// Mitsubishi GX Works2 project: Slave_V37_FERDIG   PLC: FX3U/FX3UC

// global labels: Global1
VAR_GLOBAL
  send_aapning_reg_ventil AT D8262 : INT;  (* ÅPNING REGVENTIL *)
  utstroom_analogt AT D8261 : INT;  (* FLOWMETER *)
  tanknivaa_analogt AT D8260 : INT;  (* NIVÅMÅLER *)
  start_bit AT M101 : BOOL;  (* M100 til M199 Reserveres TIL SLAVE *)
  tvangstyr_startsignal_frekv AT M1 : BOOL;  (* Aktiver kontaktor for startsignal til omformer / M0 til M99 Reservert INTERNT i slave *)
  intern_start_regventil AT M2 : BOOL;
  intern_aktiver_magventil_1 AT M4 : BOOL;  (* Lokalt for slave *)
  intern_aktiver_magventil_2 AT M5 : BOOL;  (* Lokalt for slave *)
  intern_aktiver_magventil_3 AT M6 : BOOL;  (* Lokalt for slave *)
  lest_tanknivaa AT D1 : INT;  (* LAGRING AV WORDS *)
  status_brytere AT D2 : INT;  (* Start,stopp,ACK og AutoModus *)
  referanse AT D5 : INT;
  Td AT D6 : INT;
  Ti AT D7 : INT;
  Kp AT D8 : INT;
  reg_modus AT D9 : INT;  (* 4bit *)
  u0_nompaadrag_fra_scada AT D10 : INT;
  lest_utstroom AT D21 : INT;
END_VAR
VAR_GLOBAL CONSTANT
  start_omformer : INT := 1151;  (* KONSTANTER *)
  stopp_omformer : INT := 1087;
  quickstop_omformer : INT := 1135;
  fult_aapen_regventil : INT := 4000;
  fult_lukket_regventil : INT := 500;
  fult_paadrag_pumpe : INT := 16310;  (* 16310 før skalering *)
END_VAR
VAR_GLOBAL
  fysisk_start_frekomformer AT Y000 : BOOL;  (* K4 / UTGANGER *)
  alarm_lampe AT Y001 : BOOL;  (* Alarmlampe *)
  magnetventil_1 AT Y004 : BOOL;  (* K1 *)
  magnetventil_2 AT Y005 : BOOL;  (* K2 *)
  magnetventil_3 AT Y006 : BOOL;  (* K3 *)
  strømbrudd AT M500 : BOOL;
  kritisk_refnivaa_opnaad_slave AT M202 : BOOL;
  kritiaskalarm_aapne_ventiler AT M203 : BOOL;
  kritiskalarm_nedre_stengventiler AT M206 : BOOL;
  fortsatt_kritisk_nedre AT M207 : BOOL;
  fortsatt_kritisk_oovre AT M208 : BOOL;
  fortsatt_alarm AT M209 : BOOL;
  alarm_oovre AT M300 : BOOL;  (* M300 til M399 beholdes FRA SLAVE *)
  kritiskalarm_oovre AT M301 : BOOL;
  ACK_slave AT M302 : BOOL;
  samplingstid AT D12 : INT;
  tau_lead AT D13 : INT;
  tau_lag AT D14 : INT;
  d_filter AT D15 : INT;
  rate_limit AT D16 : INT;
  tt AT D17 : INT;
  ref_skalert_som_tankmaaling AT D22 : INT;
  stasjonært_avvik AT M303 : BOOL;
END_VAR
VAR_GLOBAL CONSTANT
  hysterese_alarmgrense : INT := 20;
END_VAR
VAR_GLOBAL
  strømbrudd_slave AT M304 : BOOL;
  alarm_nedre AT M305 : BOOL;  (* M300 til M399 beholdes FRA SLAVE *)
  kritiskalarm_nedre AT M306 : BOOL;
  paadrag_manuelt AT D34 : INT;
  kritisk_lav_eller_hooy AT M210 : BOOL;
  stopp AT M201 : BOOL;
  start AT M200 : BOOL;  (* INTERNT I SLAVE *)
  oppstart AT M211 : BOOL;
  auto_ACK AT M212 : BOOL;
  stopp_slave AT M307 : BOOL;
  under_refnivaa AT M213 : BOOL;  (* M213 til M215 *)
  auto_ACK_lav_hooy AT M216 : BOOL;
  frekvenspaadrag_til_omformer AT D33 : INT;
END_VAR
VAR_GLOBAL CONSTANT
  blinkrate : INT := 1;
END_VAR
VAR_GLOBAL
  kfk AT D18 : INT;  (* Foroverkoblingsparameter *)
  forrige_paadrag_regulator AT D52 : REAL;
  tanknivaa_til_regulator AT D40 : REAL;
  u0_nompaadrag_til_regulator AT D46 : REAL;
  paadrag_fra_regulator AT D48 : REAL;
  manuelt_paadrag_til_regulator AT D50 : REAL;
  control_word AT D32 : INT;
  paadrag_til_scada AT D4 : INT;  (* Start,stopp,ACK og AutoModus *)
  tanknivaa_til_scada AT D0 : INT;
  aapning_reg_ventil AT D23 : INT;
  ventil_paadrag AT D36 : INT;
  tanknivaa_filtrert AT D24 : INT;
  stasjonært_avvik_verdi AT D25 : INT;
  paadrag_regulator AT D26 : INT;  (* RegulatorParmarametere *)
  referanse_til_PID AT D42 : REAL;
  magnetventil_1_ACK AT M308 : BOOL;
  magnetventil_2_ACK AT M309 : BOOL;
  magnetventil_3_ACK AT M310 : BOOL;
END_VAR
VAR_GLOBAL CONSTANT
  null_paadrag_pumpe : INT;  (* 16310 før skalering *)
END_VAR
VAR_GLOBAL
  glatt_referanse AT D44 : REAL;
  glatt_referanse_til_scada AT D38 : INT;
  reg_modus_bit AT M112 : BOOL;  (* Til og med M115 *)
  kritisk_lav_eller_hooy_bit AT M111 : BOOL;
  testmodus_bit AT M110 : BOOL;
  anti_windup_bit AT M109 : BOOL;
  forover_kobling_bit AT M108 : BOOL;
  pumpe_regulering_bit AT M107 : BOOL;
  ventil_regulering_bit AT M106 : BOOL;
  aktiver_magv_3_bit AT M105 : BOOL;
  aktiver_magv_2_bit AT M104 : BOOL;
  aktiver_magv_1_bit AT M103 : BOOL;
  ACK_bit AT M102 : BOOL;
  stopp_bit AT M100 : BOOL;
  magnetventil_aapen_igjen AT M311 : BOOL;
  pumpe_regulering AT M312 : BOOL;
  ventil_regulering AT M313 : BOOL;
  Profibus_ok AT M314 : BOOL;
  kritiskalarm_refnivaa_oppnaad AT M315 : BOOL;
  ventil_skalert AT D37 : INT;
  utstroom_filtrert AT D20 : INT;
  frk_control AT M400 : BOOL;  (* Høy = klar, Lav = ikke klar / Statusmeldinger fra frekvensomformeren *)
  frk_VLT AT M401 : BOOL;
  frk_motor_coasting AT M402 : BOOL;
  frk_trip AT M403 : BOOL;
  frk_on_2 AT M404 : BOOL;
  frk_on_3 AT M405 : BOOL;
  frk_stop_enable AT M406 : BOOL;
  frk_warning AT M407 : BOOL;
  frk_speed_ref AT M408 : BOOL;
  frk_local_operation AT M409 : BOOL;
  frk_frequency_ok AT M410 : BOOL;
  frk_running AT M411 : BOOL;
  frk_spenning_ok AT M413 : BOOL;
  frk_moment_ok AT M414 : BOOL;
  frk_termisk_varsel AT M415 : BOOL;
  testmode_ACK AT M316 : BOOL;
  utstroom_til_regulator AT D54 : REAL;
  utstroom_til_scada AT D39 : INT;
  ubrukt_2 AT D100 : INT;
  ubrukt_3 AT D101 : INT;
  ubrukt_4 AT D102 : INT;
  ubrukt_15 AT D103 : INT;
  innenfor_refomraade AT M214 : BOOL;  (* M213 til M215 *)
  over_refnivaa AT M215 : BOOL;  (* M213 til M215 *)
  reg_modus_ACK AT M317 : BOOL;  (* M317 til og med M320 *)
  under_60_nivaa AT M217 : BOOL;
  frekvens_skalert AT D35 : INT;
END_VAR

// task Task_01 (event TRUE, interval 0, priority 31): POU_01
// task task_2 (event FALSE, interval T#200ms, priority 31): Regulator
// task stroombrudd (event TRUE, interval 0, priority 31): stroombrudd

PROGRAM POU_01
VAR
  lavpass_filter_1 : lavpass_filter_tanknivaa;
  lavpass_filter_2 : lavpass_filter_utstrøm;
  DEROUND_1 : DEROUND;
  DEROUND_2 : DEROUND;
  Lampe_Alarm_1 : Lampe_Alarm;
  DEROUND_3 : DEROUND;
  DEROUND_4 : DEROUND;
  DEROUND_5 : DEROUND;
  DEROUND_6 : DEROUND;
  DEROUND_7 : DEROUND;
  skalering_tanknivaa_1 : skalering_tanknivaa;
  skalering_ventil_1 : skalering_ventil;
  skalering_paadrag_1 : skalering_paadrag;
  skalering_referanse_1 : skalering_referanse;
  utregning_stasjonært_avvik_1 : utregning_stasjonært_avvik;
  skalering_til_bruker_ven_og_omf1 : skalering_til_bruker_ven_og_omf;
  skalering_utstroom_1 : skalering_utstroom;
  mottak_av_data_fra_master_1 : mottak_av_data_fra_master;
  sending_av_data_til_master_1 : sending_av_data_til_master;
  kvittering_av_alarmer_1 : kvittering_av_alarmer;
  utganger_1 : utganger;
  kritisk_refnivaa_oppnaad_1 : kritisk_refnivaa_oppnaad;
  reguleringsmodus_1 : reguleringsmodus;
  handling_ved_kritisk_alarm_1 : handling_ved_kritisk_alarm;
  alarmgrenser_1 : alarmgrenser;
END_VAR
(* structured ladder/FBD written out as ST: instructions are called as NAME(EN, inputs, outputs); _pN, _eN, _tN stand for wires *)
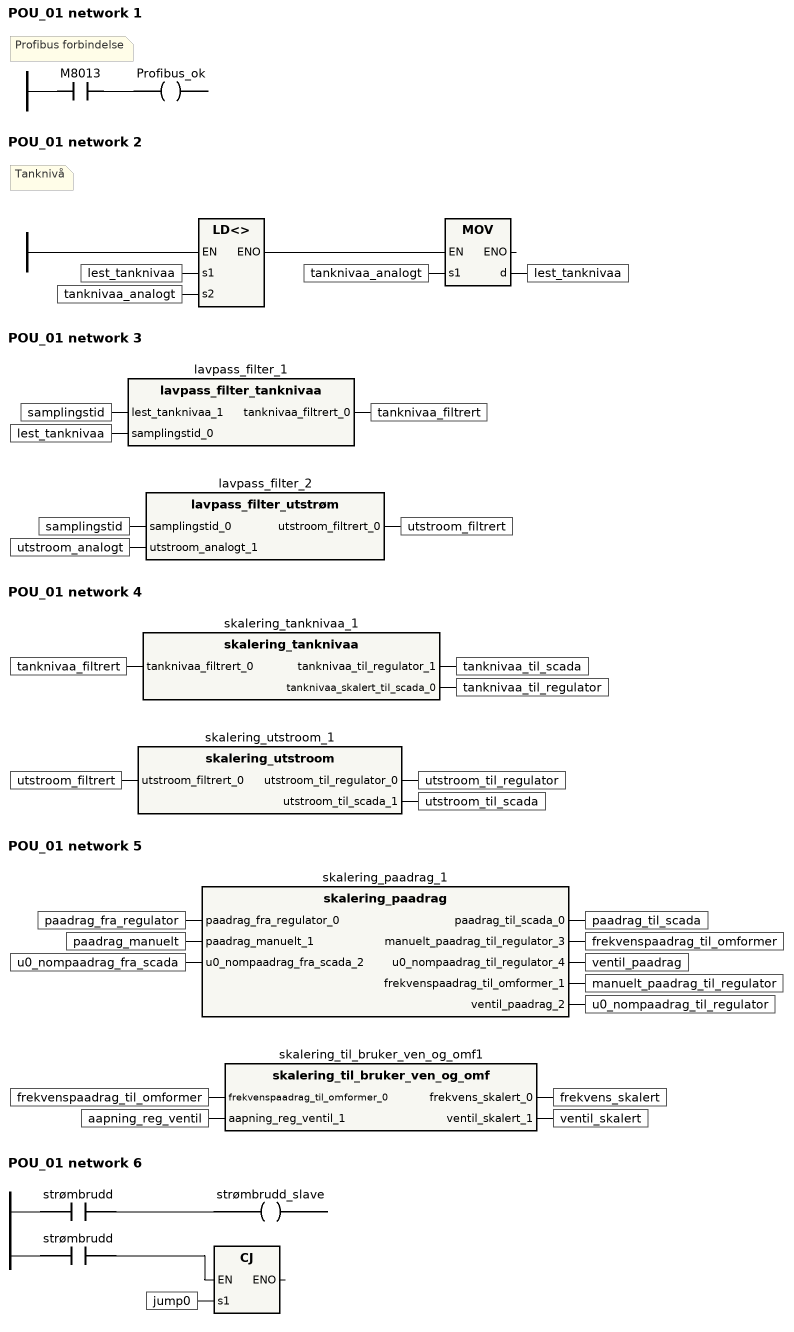
(* network 1 *)
(* Profibus forbindelse *)
Profibus_ok := M8013;
(* network 2 *)
(* Tanknivå *)
_e1 := LD<>(TRUE, lest_tanknivaa, tanknivaa_analogt);
MOV(_e1, tanknivaa_analogt, lest_tanknivaa);
(* network 3 *)
lavpass_filter_1(lest_tanknivaa_1 := samplingstid, samplingstid_0 := lest_tanknivaa, tanknivaa_filtrert_0 => tanknivaa_filtrert);
lavpass_filter_2(samplingstid_0 := samplingstid, utstroom_analogt_1 := utstroom_analogt, utstroom_filtrert_0 => utstroom_filtrert);
(* network 4 *)
skalering_tanknivaa_1(tanknivaa_filtrert_0 := tanknivaa_filtrert, tanknivaa_til_regulator_1 => tanknivaa_til_scada, tanknivaa_skalert_til_scada_0 => tanknivaa_til_regulator);
skalering_utstroom_1(utstroom_filtrert_0 := utstroom_filtrert, utstroom_til_regulator_0 => utstroom_til_regulator, utstroom_til_scada_1 => utstroom_til_scada);
(* network 5 *)
skalering_paadrag_1(paadrag_fra_regulator_0 := paadrag_fra_regulator, paadrag_manuelt_1 := paadrag_manuelt, u0_nompaadrag_fra_scada_2 := u0_nompaadrag_fra_scada, paadrag_til_scada_0 => paadrag_til_scada, manuelt_paadrag_til_regulator_3 => frekvenspaadrag_til_omformer, u0_nompaadrag_til_regulator_4 => ventil_paadrag, frekvenspaadrag_til_omformer_1 => manuelt_paadrag_til_regulator, ventil_paadrag_2 => u0_nompaadrag_til_regulator);
skalering_til_bruker_ven_og_omf1(frekvenspaadrag_til_omformer_0 := frekvenspaadrag_til_omformer, aapning_reg_ventil_1 := aapning_reg_ventil, frekvens_skalert_0 => frekvens_skalert, ventil_skalert_1 => ventil_skalert);
(* network 6 *)
strømbrudd_slave := strømbrudd;
CJ(strømbrudd, jump0);
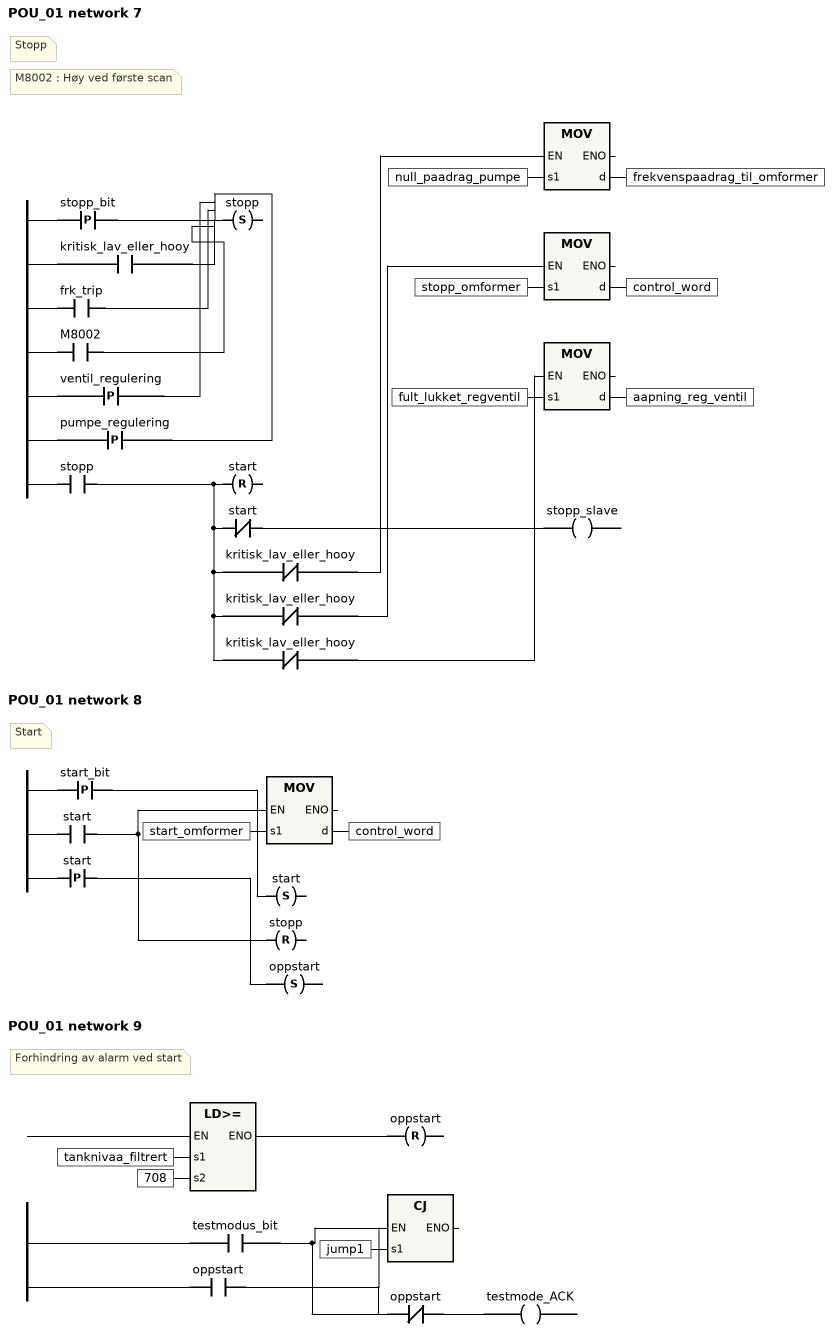
(* network 7 *)
(* Stopp *)
(* M8002 : Høy ved første scan *)
SET(LDP(TRUE, stopp_bit) OR kritisk_lav_eller_hooy OR frk_trip OR M8002 OR LDP(TRUE, ventil_regulering) OR LDP(TRUE, pumpe_regulering), stopp);
RST(stopp, start);
stopp_slave := stopp AND NOT start;
MOV(stopp AND NOT kritisk_lav_eller_hooy, null_paadrag_pumpe, frekvenspaadrag_til_omformer);
MOV(stopp AND NOT kritisk_lav_eller_hooy, stopp_omformer, control_word);
MOV(stopp AND NOT kritisk_lav_eller_hooy, fult_lukket_regventil, aapning_reg_ventil);
(* network 8 *)
(* Start *)
SET(LDP(TRUE, start_bit), start);
RST(start, stopp);
MOV(start, start_omformer, control_word);
SET(LDP(TRUE, start), oppstart);
(* network 9 *)
(* Forhindring av alarm ved start *)
_e1 := LD>=(TRUE, tanknivaa_filtrert, 708);
RST(_e1, oppstart);
_p2 := testmodus_bit OR oppstart;
testmode_ACK := _p2 AND NOT oppstart;
CJ(_p2, jump1);
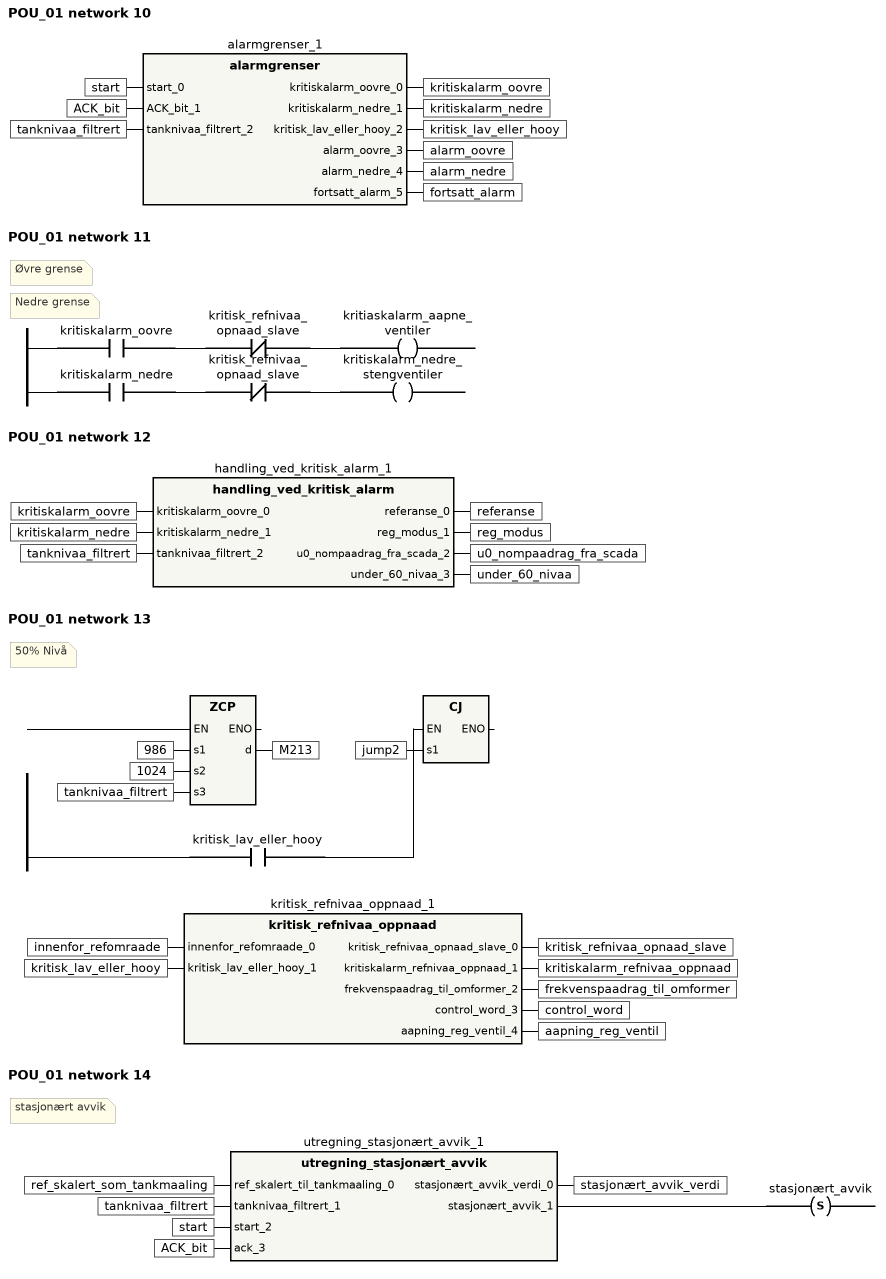
(* network 10 *)
alarmgrenser_1(start_0 := start, ACK_bit_1 := ACK_bit, tanknivaa_filtrert_2 := tanknivaa_filtrert, kritiskalarm_oovre_0 => kritiskalarm_oovre, kritiskalarm_nedre_1 => kritiskalarm_nedre, kritisk_lav_eller_hooy_2 => kritisk_lav_eller_hooy, alarm_oovre_3 => alarm_oovre, alarm_nedre_4 => alarm_nedre, fortsatt_alarm_5 => fortsatt_alarm);
(* network 11 *)
(* Øvre grense *)
(* Nedre grense *)
kritiaskalarm_aapne_ventiler := kritiskalarm_oovre AND NOT kritisk_refnivaa_opnaad_slave;
kritiskalarm_nedre_stengventiler := kritiskalarm_nedre AND NOT kritisk_refnivaa_opnaad_slave;
(* network 12 *)
handling_ved_kritisk_alarm_1(kritiskalarm_oovre_0 := kritiskalarm_oovre, kritiskalarm_nedre_1 := kritiskalarm_nedre, tanknivaa_filtrert_2 := tanknivaa_filtrert, referanse_0 => referanse, reg_modus_1 => reg_modus, u0_nompaadrag_fra_scada_2 => u0_nompaadrag_fra_scada, under_60_nivaa_3 => under_60_nivaa);
(* network 13 *)
(* 50% Nivå *)
ZCP(TRUE, 986, 1024, tanknivaa_filtrert, M213);
kritisk_refnivaa_oppnaad_1(innenfor_refomraade_0 := innenfor_refomraade, kritisk_lav_eller_hooy_1 := kritisk_lav_eller_hooy, kritisk_refnivaa_opnaad_slave_0 => kritisk_refnivaa_opnaad_slave, kritiskalarm_refnivaa_oppnaad_1 => kritiskalarm_refnivaa_oppnaad, frekvenspaadrag_til_omformer_2 => frekvenspaadrag_til_omformer, control_word_3 => control_word, aapning_reg_ventil_4 => aapning_reg_ventil);
CJ(kritisk_lav_eller_hooy, jump2);
(* network 14 *)
(* stasjonært avvik *)
utregning_stasjonært_avvik_1(ref_skalert_til_tankmaaling_0 := ref_skalert_som_tankmaaling, tanknivaa_filtrert_1 := tanknivaa_filtrert, start_2 := start, ack_3 := ACK_bit, stasjonært_avvik_verdi_0 => stasjonært_avvik_verdi);
SET(utregning_stasjonært_avvik_1.stasjonært_avvik_1, stasjonært_avvik);
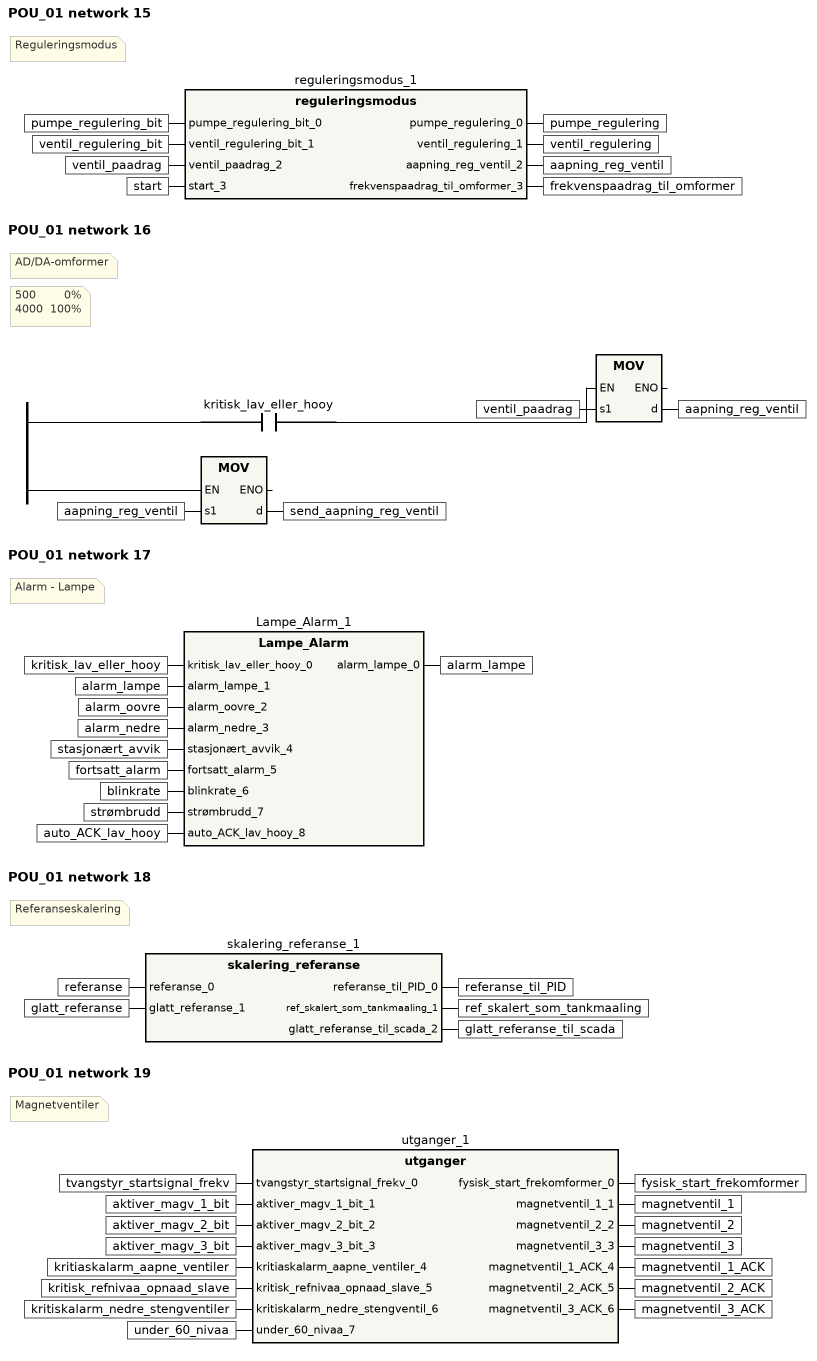
(* network 15 jump1: *)
(* Reguleringsmodus *)
reguleringsmodus_1(pumpe_regulering_bit_0 := pumpe_regulering_bit, ventil_regulering_bit_1 := ventil_regulering_bit, ventil_paadrag_2 := ventil_paadrag, start_3 := start, pumpe_regulering_0 => pumpe_regulering, ventil_regulering_1 => ventil_regulering, aapning_reg_ventil_2 => aapning_reg_ventil, frekvenspaadrag_til_omformer_3 => frekvenspaadrag_til_omformer);
(* network 16 jump2: *)
(* AD/DA-omformer *)
(* 500        0% / 4000  100% *)
MOV(kritisk_lav_eller_hooy, ventil_paadrag, aapning_reg_ventil);
MOV(TRUE, aapning_reg_ventil, send_aapning_reg_ventil);
(* network 17 *)
(* Alarm - Lampe *)
Lampe_Alarm_1(kritisk_lav_eller_hooy_0 := kritisk_lav_eller_hooy, alarm_lampe_1 := alarm_lampe, alarm_oovre_2 := alarm_oovre, alarm_nedre_3 := alarm_nedre, stasjonært_avvik_4 := stasjonært_avvik, fortsatt_alarm_5 := fortsatt_alarm, blinkrate_6 := blinkrate, strømbrudd_7 := strømbrudd, auto_ACK_lav_hooy_8 := auto_ACK_lav_hooy, alarm_lampe_0 => alarm_lampe);
(* network 18 *)
(* Referanseskalering *)
skalering_referanse_1(referanse_0 := referanse, glatt_referanse_1 := glatt_referanse, referanse_til_PID_0 => referanse_til_PID, ref_skalert_som_tankmaaling_1 => ref_skalert_som_tankmaaling, glatt_referanse_til_scada_2 => glatt_referanse_til_scada);
(* network 19 *)
(* Magnetventiler *)
utganger_1(tvangstyr_startsignal_frekv_0 := tvangstyr_startsignal_frekv, aktiver_magv_1_bit_1 := aktiver_magv_1_bit, aktiver_magv_2_bit_2 := aktiver_magv_2_bit, aktiver_magv_3_bit_3 := aktiver_magv_3_bit, kritiaskalarm_aapne_ventiler_4 := kritiaskalarm_aapne_ventiler, kritisk_refnivaa_opnaad_slave_5 := kritisk_refnivaa_opnaad_slave, kritiskalarm_nedre_stengventil_6 := kritiskalarm_nedre_stengventiler, under_60_nivaa_7 := under_60_nivaa, fysisk_start_frekomformer_0 => fysisk_start_frekomformer, magnetventil_1_1 => magnetventil_1, magnetventil_2_2 => magnetventil_2, magnetventil_3_3 => magnetventil_3, magnetventil_1_ACK_4 => magnetventil_1_ACK, magnetventil_2_ACK_5 => magnetventil_2_ACK, magnetventil_3_ACK_6 => magnetventil_3_ACK);
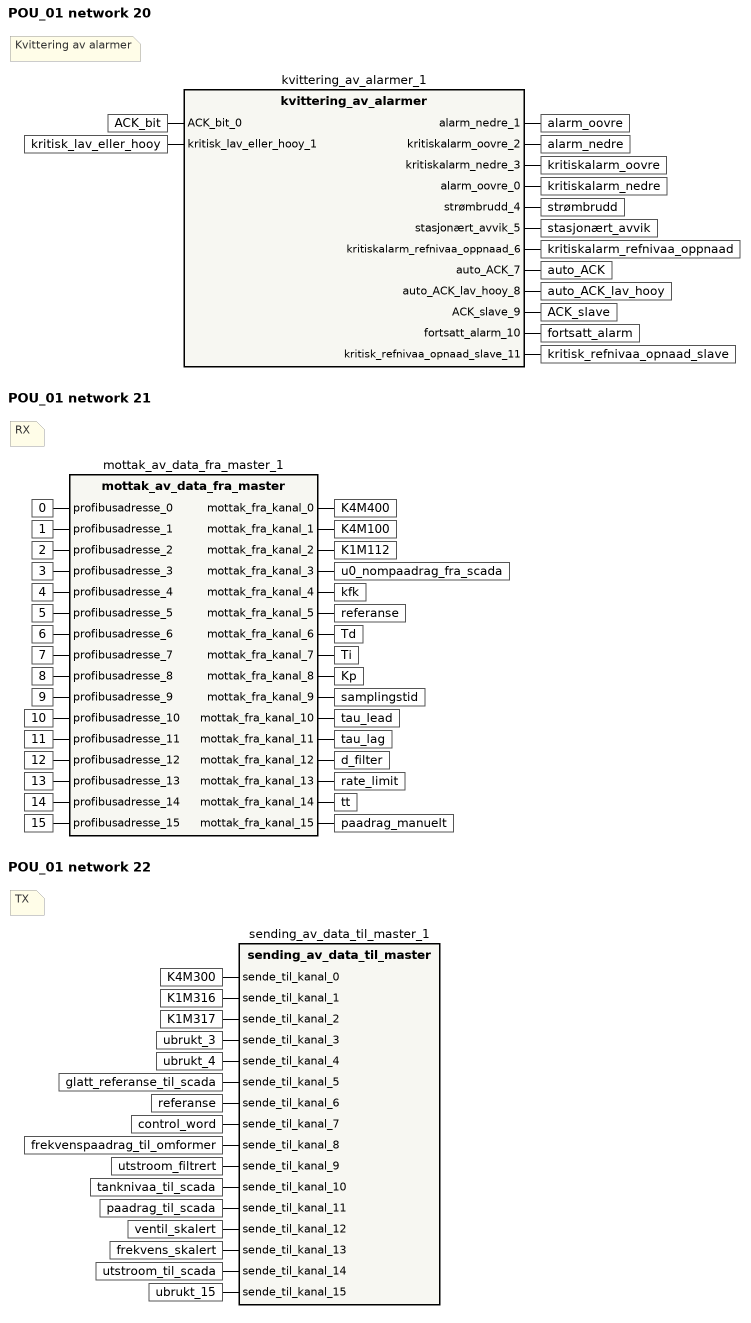
(* network 20 jump0: *)
(* Kvittering av alarmer *)
kvittering_av_alarmer_1(ACK_bit_0 := ACK_bit, kritisk_lav_eller_hooy_1 := kritisk_lav_eller_hooy, alarm_nedre_1 => alarm_oovre, kritiskalarm_oovre_2 => alarm_nedre, kritiskalarm_nedre_3 => kritiskalarm_oovre, alarm_oovre_0 => kritiskalarm_nedre, strømbrudd_4 => strømbrudd, stasjonært_avvik_5 => stasjonært_avvik, kritiskalarm_refnivaa_oppnaad_6 => kritiskalarm_refnivaa_oppnaad, auto_ACK_7 => auto_ACK, auto_ACK_lav_hooy_8 => auto_ACK_lav_hooy, ACK_slave_9 => ACK_slave, fortsatt_alarm_10 => fortsatt_alarm, kritisk_refnivaa_opnaad_slave_11 => kritisk_refnivaa_opnaad_slave);
(* network 21 *)
(* RX *)
mottak_av_data_fra_master_1(profibusadresse_0 := 0, profibusadresse_1 := 1, profibusadresse_2 := 2, profibusadresse_3 := 3, profibusadresse_4 := 4, profibusadresse_5 := 5, profibusadresse_6 := 6, profibusadresse_7 := 7, profibusadresse_8 := 8, profibusadresse_9 := 9, profibusadresse_10 := 10, profibusadresse_11 := 11, profibusadresse_12 := 12, profibusadresse_13 := 13, profibusadresse_14 := 14, profibusadresse_15 := 15, mottak_fra_kanal_0 => K4M400, mottak_fra_kanal_1 => K4M100, mottak_fra_kanal_2 => K1M112, mottak_fra_kanal_3 => u0_nompaadrag_fra_scada, mottak_fra_kanal_4 => kfk, mottak_fra_kanal_5 => referanse, mottak_fra_kanal_6 => Td, mottak_fra_kanal_7 => Ti, mottak_fra_kanal_8 => Kp, mottak_fra_kanal_9 => samplingstid, mottak_fra_kanal_10 => tau_lead, mottak_fra_kanal_11 => tau_lag, mottak_fra_kanal_12 => d_filter, mottak_fra_kanal_13 => rate_limit, mottak_fra_kanal_14 => tt, mottak_fra_kanal_15 => paadrag_manuelt);
(* network 22 *)
(* TX *)
sending_av_data_til_master_1(sende_til_kanal_0 := K4M300, sende_til_kanal_1 := K1M316, sende_til_kanal_2 := K1M317, sende_til_kanal_3 := ubrukt_3, sende_til_kanal_4 := ubrukt_4, sende_til_kanal_5 := glatt_referanse_til_scada, sende_til_kanal_6 := referanse, sende_til_kanal_7 := control_word, sende_til_kanal_8 := frekvenspaadrag_til_omformer, sende_til_kanal_9 := utstroom_filtrert, sende_til_kanal_10 := tanknivaa_til_scada, sende_til_kanal_11 := paadrag_til_scada, sende_til_kanal_12 := ventil_skalert, sende_til_kanal_13 := frekvens_skalert, sende_til_kanal_14 := utstroom_til_scada, sende_til_kanal_15 := ubrukt_15);
END_PROGRAM

FUNCTION_BLOCK lavpass_filter_tanknivaa
VAR CONSTANT
  omega_0 : REAL := 0.2;  (* cutoff frekvens. 16.4: 0.25 mye støy?? gamle:0.0384 *)
  two_pi : REAL := 6.28;  (* 2*pi *)
END_VAR
VAR
  input_float : REAL;
  avg_maaling : REAL;
  avg_maaling_k_minus_1 : REAL;
  filter_faktor : REAL;
  eksponent : REAL;
  tastetid_float : REAL;
END_VAR
VAR_INPUT
  lest_tanknivaa_1 : INT;
END_VAR
VAR_OUTPUT
  tanknivaa_filtrert_0 : INT;
END_VAR
VAR_INPUT
  samplingstid_0 : INT;
END_VAR
VAR
  DEROUND_1 : DEROUND;
END_VAR
tastetid_float :=  INT_TO_REAL (samplingstid_0)/100.0;
eksponent := -tastetid_float*omega_0*two_pi;
filter_faktor := EXP(eksponent);
input_float := INT_TO_REAL (lest_tanknivaa_1);
avg_maaling := filter_faktor * avg_maaling_k_minus_1 + (1.0 - filter_faktor) * input_float;
avg_maaling_k_minus_1 := avg_maaling;
DEROUND_1(real_to_round := avg_maaling, gjelende_siffer_input := 0);
tanknivaa_filtrert_0 := REAL_TO_INT(DEROUND_1.real_rounded);
END_FUNCTION_BLOCK

FUNCTION_BLOCK DEROUND
VAR_INPUT
  real_to_round : REAL;
  gjelende_siffer_input : INT;
END_VAR
VAR
  gjelende_siffer_real : REAL;
  ti_til_gjellende_siffer : REAL;
  int_round : DINT;
END_VAR
VAR_OUTPUT
  real_rounded : REAL;
END_VAR
gjelende_siffer_real := INT_TO_REAL(gjelende_siffer_input);
ti_til_gjellende_siffer := EXP(gjelende_siffer_real * LN(10.0));

IF DINT_TO_REAL(REAL_TO_DINT(real_to_round* ti_til_gjellende_siffer) ) > (real_to_round*ti_til_gjellende_siffer - 0.5) THEN;
	int_round := REAL_TO_DINT(real_to_round * ti_til_gjellende_siffer);
	real_rounded := DINT_TO_REAL(int_round)/ti_til_gjellende_siffer;
ELSE
	int_round := REAL_TO_DINT(real_to_round * ti_til_gjellende_siffer + 1.0);
	real_rounded := DINT_TO_REAL(int_round)/ti_til_gjellende_siffer;
END_IF;
END_FUNCTION_BLOCK

FUNCTION_BLOCK Lampe_Alarm
VAR_OUTPUT
  alarm_lampe_0 : BOOL;
END_VAR
VAR_INPUT
  kritisk_lav_eller_hooy_0 : BOOL;
  alarm_lampe_1 : BOOL;
  alarm_oovre_2 : BOOL;
  alarm_nedre_3 : BOOL;
  stasjonært_avvik_4 : BOOL;
  fortsatt_alarm_5 : BOOL;
  blinkrate_6 : INT;
  strømbrudd_7 : BOOL;
  auto_ACK_lav_hooy_8 : BOOL;
END_VAR
VAR
  lampe_5HZ : BOOL;
  lampe_1HZ : BOOL;
  lampe_konstant : BOOL;
END_VAR
(* structured ladder/FBD written out as ST: instructions are called as NAME(EN, inputs, outputs); _pN, _eN, _tN stand for wires *)
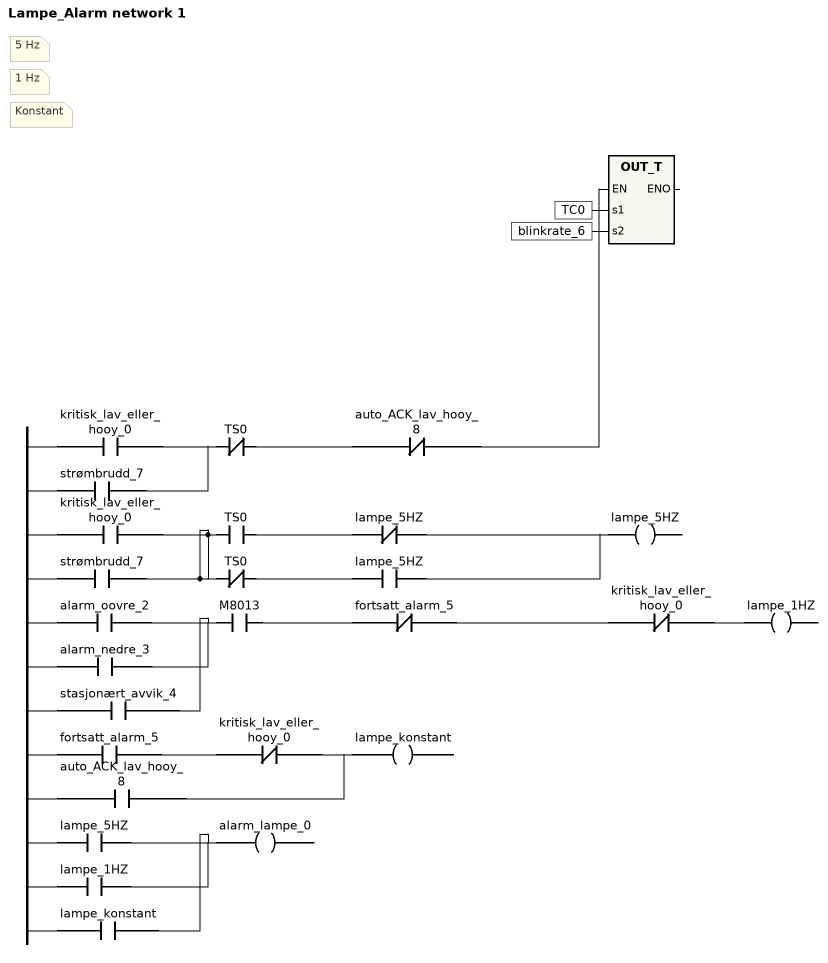
(* network 1 *)
(* 5 Hz *)
(* 1 Hz *)
(* Konstant *)
OUT_T(((kritisk_lav_eller_hooy_0 OR strømbrudd_7) AND NOT TS0) AND NOT auto_ACK_lav_hooy_8, TC0, blinkrate_6);
_p1 := kritisk_lav_eller_hooy_0 OR strømbrudd_7;
lampe_5HZ := (_p1 AND TS0 AND NOT lampe_5HZ) OR (_p1 AND NOT TS0 AND lampe_5HZ);
lampe_1HZ := (((alarm_oovre_2 OR alarm_nedre_3 OR stasjonært_avvik_4) AND M8013) AND NOT fortsatt_alarm_5) AND NOT kritisk_lav_eller_hooy_0;
lampe_konstant := (fortsatt_alarm_5 AND NOT kritisk_lav_eller_hooy_0) OR auto_ACK_lav_hooy_8;
alarm_lampe_0 := lampe_5HZ OR lampe_1HZ OR lampe_konstant;
END_FUNCTION_BLOCK

FUNCTION_BLOCK Lead_lag
VAR_OUTPUT
  u_fk : REAL;
END_VAR
VAR_INPUT
  Kf : INT;  (* random konstant per nå *)
END_VAR
VAR
  forstyrr : REAL;  (* forstyrrelse *)
END_VAR
VAR_INPUT
  Tlead : INT;  (* random konstant per nå *)
  Tlag : INT;  (* random konstant per nå *)
END_VAR
VAR
  last_v : REAL;
END_VAR
VAR_INPUT
  Ts : INT;
END_VAR
VAR
  last_u_fk : REAL;
END_VAR
VAR_INPUT
  leadlag : BOOL;
END_VAR
VAR
  Kf_ny : REAL;
  Tlead_ny : REAL;
  Tlag_ny : REAL;
  Ts_ut : REAL;
END_VAR
VAR_INPUT
  reset : BOOL;
  y_1 : REAL;
  outflow : REAL;
END_VAR
VAR
  forstyrr_ny : REAL;
END_VAR
IF (reset) THEN
	last_v := 0.0;
	last_u_fk := 0.0;
END_IF;

(*Trengs det skalering??*)
Kf_ny := INT_TO_REAL(Kf)/100.00;
Tlead_ny := INT_TO_REAL(Tlead)/100.00;
Tlag_ny := INT_TO_REAL(Tlag)/100.00;
Ts_ut := INT_TO_REAL(Ts)/100.00;

forstyrr := outflow - 0.00025367*y_1*y_1*y_1+0.04313578*y_1*y_1-2.8730536*y_1-5.08111888;

IF forstyrr < 0.00 THEN
	forstyrr_ny := 0.00;
ELSE
	forstyrr_ny := forstyrr;
END_IF;


IF (leadlag=1) THEN
	u_fk := (Kf_ny*Tlead_ny*(forstyrr_ny-last_v)+Kf_ny*forstyrr_ny*Ts_ut+Tlag_ny*last_u_fk)/(Ts_ut+Tlag_ny); 
	(*ingen tidsforsinkelse her, skal vi ha det??*)
	last_v := forstyrr_ny;
	last_u_fk := u_fk;
ELSE
	u_fk := 0.00;
	last_u_fk := 0.00;
END_IF;
END_FUNCTION_BLOCK

FUNCTION_BLOCK PID_regulator
VAR
  last_y : REAL;
END_VAR
VAR_INPUT
  Ts : INT;  (* 0.04 *)
END_VAR
VAR
  up : REAL;
  ud : REAL;
END_VAR
VAR_OUTPUT
  ui : REAL;
END_VAR
VAR
  e_reg : REAL;
  alpha : REAL;
  beta : REAL;
  last_ui : REAL;
  last_ud : REAL;
  last_up : REAL;
END_VAR
VAR_INPUT
  ni : INT;  (* mulig dette skal være input fra intouch idk. *)
  Kp_reg : INT;
  Ti_reg : INT;
  Td_reg : INT;
  r_1 : REAL;
END_VAR
VAR_OUTPUT
  u_ut : REAL;  (* endre til word *)
END_VAR
VAR_INPUT
  y_1 : REAL;
  manual_input : REAL;  (* endre til word *)
  Regulator_type : INT;
  u_fk : REAL;
  u_antiwindup : REAL;
END_VAR
VAR
  Kp_ut : REAL;
  Ti_ut : REAL;
  Td_ut : REAL;
END_VAR
VAR_OUTPUT
  last_u : REAL;
END_VAR
VAR_INPUT
  ratebegrensing : INT;  (* initial value = 2 *)
END_VAR
VAR
  Ts_ut : REAL;
  d_filt : REAL;
  u_reg : REAL;
END_VAR
VAR_INPUT
  reset : BOOL;
  u_it : REAL;
END_VAR
VAR_OUTPUT
  u_t : REAL;
END_VAR
VAR_INPUT
  u_rykkfri : REAL;
END_VAR
VAR
  last_u_nom : REAL;
END_VAR
VAR_INPUT
  u_nominel : REAL;
END_VAR
VAR
  u_nom : REAL;
  konstant : REAL;
END_VAR
IF (reset) THEN
	last_up := 0.0;
	last_ui := 0.0;
	last_ud := 0.0;
	last_y := 0.0;
	last_u_nom := 0.00;
END_IF;

Kp_ut := INT_TO_REAL(Kp)/100.00;
Ti_ut := INT_TO_REAL(Ti)/100.00; 
Td_ut := INT_TO_REAL(Td)/100.00;
Ts_ut := INT_TO_REAL(Ts)/100.00;
d_filt := INT_TO_REAL(ni)/100.00; 

e_reg := r_1-y_1;

alpha := Ts_ut / Ti_ut;
beta :=  Td_ut/(Td_ut+d_filt*Ts_ut);

up := e_reg*Kp_ut;

IF (up-last_up>INT_TO_REAL(ratebegrensing)) THEN
	up := last_up+INT_TO_REAL(ratebegrensing);
ELSIF (up-last_up<INT_TO_REAL(0-ratebegrensing)) THEN
	up := last_up - INT_TO_REAL(ratebegrensing);
END_IF;

IF (e_reg)<0.00 THEN
	konstant := 1.00;
ELSE
	konstant := 1.00;
END_IF;

ui := last_ui + Kp_ut*alpha* e_reg*konstant+u_it+u_antiwindup;

IF (ui-last_ui>INT_TO_REAL(ratebegrensing)) THEN
	ui := last_ui+INT_TO_REAL(ratebegrensing);
ELSIF (ui-last_ui<INT_TO_REAL(0-ratebegrensing)) THEN
	ui := last_ui - INT_TO_REAL(ratebegrensing);
END_IF;

ud := beta*last_ud-Kp_ut*(Td_ut/Ts_ut)*(1.00-beta)*(y_1-last_y);

IF (ud-last_ud>INT_TO_REAL(ratebegrensing)) THEN
	ud := last_ud+INT_TO_REAL(ratebegrensing);
ELSIF (ud-last_ud<INT_TO_REAL(0-ratebegrensing)) THEN
	ud := last_ud - INT_TO_REAL(ratebegrensing);
END_IF;

(*velger regulatortype*)
CASE regulator_type OF
	0: 
	u_reg := manual_input;
	ui := 0.00;
(*	up := 0.00;
	ud := 0.00;*)
	1: 
	u_reg := up+u_nominel+u_fk+u_rykkfri;
	ui := u_nominel;
(*	ud := 0.00;*)
	2: 
	u_reg := up+ui+u_fk+u_rykkfri;
	(*ud := 0.00;*)
	3: 
	u_reg := up+ud+u_nominel+u_fk+u_rykkfri;
	ui := u_nominel;
	4: 
	u_reg := up+ui+ud+u_fk+u_rykkfri;
END_CASE;

u_t := u_reg;

IF u_reg<0.00 THEN
	u_reg := 0.00;
END_IF;

IF (u_reg-last_u>INT_TO_REAL(ratebegrensing)) THEN
	u_reg := last_u+INT_TO_REAL(ratebegrensing);
ELSIF (u_reg-last_u<INT_TO_REAL(0-ratebegrensing)) THEN
	u_reg := last_u - INT_TO_REAL(ratebegrensing);
END_IF;

u_nom := u_nominel;

IF (u_nominel-last_u_nom>INT_TO_REAL(ratebegrensing)) THEN
	u_nom := last_u_nom+INT_TO_REAL(ratebegrensing);
ELSIF (u_nominel-last_u_nom<INT_TO_REAL(0-ratebegrensing)) THEN
	u_nom := last_u_nom - INT_TO_REAL(ratebegrensing);
END_IF;

last_u_nom := u_nom;
last_u := u_reg;
last_up := up;
last_ui := ui;
last_ud := ud;
last_y :=  y_1;
u_ut := u_reg;
END_FUNCTION_BLOCK

FUNCTION_BLOCK Referanseglatter
VAR_INPUT
  r_inn : REAL;
END_VAR
VAR_OUTPUT
  referanse_ut : REAL;
END_VAR
VAR CONSTANT
  a_rglatt : REAL := 5;
  b : REAL := 4.47;
END_VAR
VAR_INPUT
  Ts : INT;
END_VAR
VAR
  Ts_ut : REAL;
  r_glatting : REAL;
  last_rut : REAL;
  lastlast_rut : REAL;
END_VAR
IF (M8002) THEN
	last_rut := 0.0;
	lastlast_rut := 0.0;
END_IF;

Ts_ut := INT_TO_REAL(Ts)/100.00;
r_glatting := r_inn;

referanse_ut := (Ts_ut*Ts_ut*a_rglatt*r_glatting-lastlast_rut+(2.00+b*Ts_ut)*last_rut)/(1.00+Ts_ut*b+a_rglatt*Ts_ut*Ts_ut);

lastlast_rut := last_rut;
last_rut := referanse_ut;
END_FUNCTION_BLOCK

FUNCTION_BLOCK Tracking
VAR_INPUT
  u_t : REAL;
END_VAR
VAR CONSTANT
  u_metning : REAL := 100.00;  (* random konstant per nå *)
END_VAR
VAR
  u_aw : REAL;
  last_u_antiwindup : REAL;
END_VAR
VAR_OUTPUT
  u_antiwindup : REAL;
END_VAR
VAR_INPUT
  Ts : INT;
  T_tracking : INT;  (* default: 0.87 *)
  last_u : REAL;
END_VAR
VAR
  u_rf : REAL;
END_VAR
VAR_INPUT
  aw_på : BOOL;
END_VAR
VAR
  Ts_ut : REAL;
  T_tut : REAL;
END_VAR
VAR_INPUT
  reset : BOOL;
  ui : REAL;
END_VAR
VAR_OUTPUT
  u_it : REAL;
END_VAR
VAR
  last_u_it : REAL;
END_VAR
VAR_OUTPUT
  u_rykkfri : REAL;
END_VAR
VAR
  last_u_rykkfri : REAL;
END_VAR
IF (reset) THEN;
	last_u_antiwindup := 0.00;
	last_u_rykkfri := 0.00;
END_IF;

Ts_ut := INT_TO_REAL(Ts)/100.00;
T_tut := INT_TO_REAL(T_tracking)/100.00;

u_aw := u_metning-u_t;
u_rf := u_t;  

IF ((u_aw+5.00)<0.00) THEN;
	IF (aw_på) THEN;
		u_antiwindup := u_aw*(Ts_ut/T_tut)+last_u_antiwindup;
	ELSE;
		u_antiwindup := 0.00;
	END_IF;
ELSIF (u_t<0.00) THEN;
	IF (aw_på) THEN;
		u_antiwindup := -u_t*(Ts_ut/T_tut)+last_u_antiwindup;
	ELSE;
		u_antiwindup := 0.00;
	END_IF;
ELSIF((u_rf+10.00)<last_u) THEN;
	u_rykkfri := (last_u-u_rf)*(Ts_ut/T_tut)+last_u_rykkfri;
ELSIF((u_rf-10.00)>last_u) THEN;
	u_rykkfri := (last_u-u_rf)*(Ts_ut/T_tut)+last_u_rykkfri;
ELSE;
	u_rykkfri := 0.00;
	u_antiwindup := 0.00;
END_IF;

last_u_antiwindup := u_antiwindup;
last_u_rykkfri := u_rykkfri;
END_FUNCTION_BLOCK

PROGRAM Regulator
VAR
  Lead_lag_1 : Lead_lag;
  Tracking_1 : Tracking;
  PID_regulator_1 : PID_regulator;
  Referanseglatter_1 : Referanseglatter;
  resettverdier : BOOL;
  integralledd : REAL;
  uit : REAL;
  ut : REAL;
END_VAR
(* structured ladder/FBD written out as ST: instructions are called as NAME(EN, inputs, outputs); _pN, _eN, _tN stand for wires *)
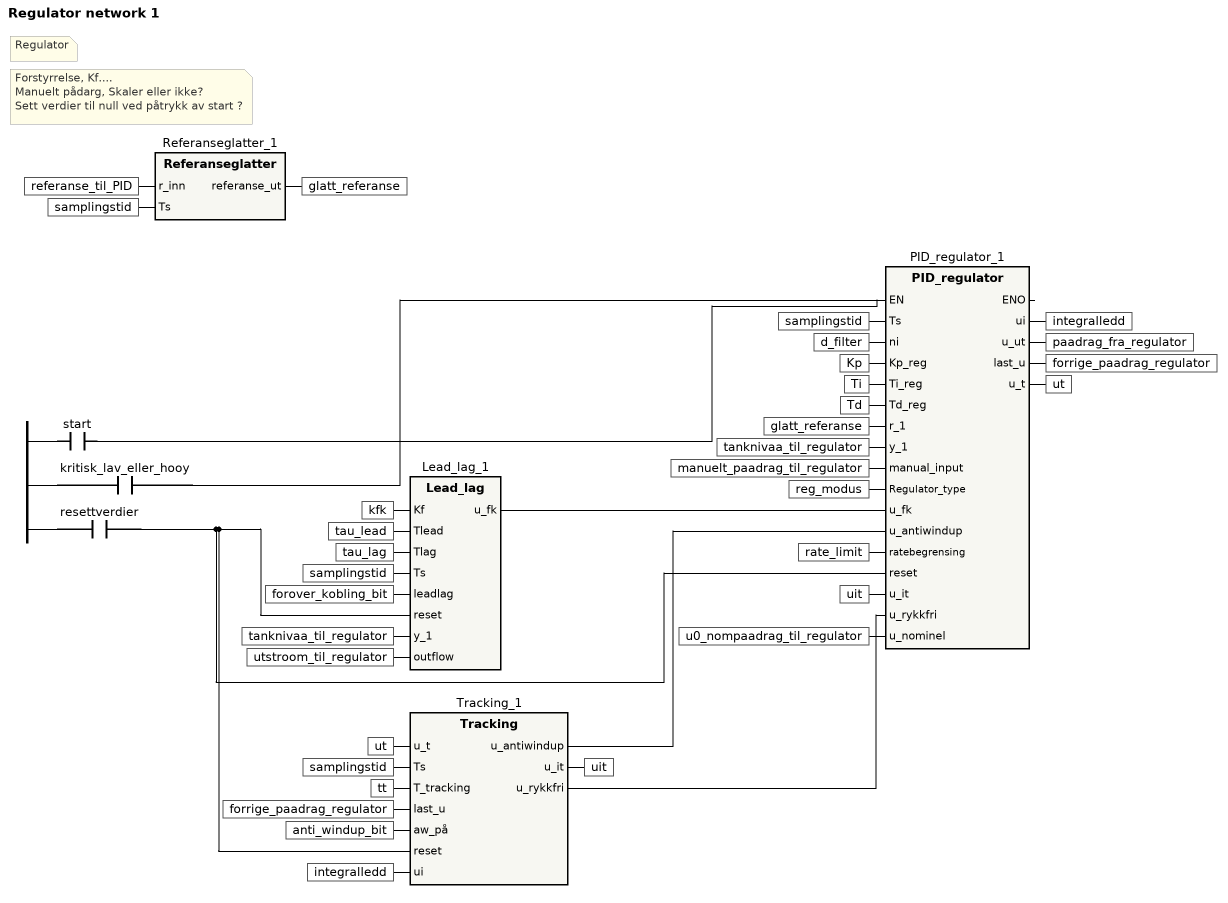
(* network 1 *)
(* Regulator *)
(* Forstyrrelse, Kf.... /  / Manuelt pådarg, Skaler eller ikke? /  / Sett verdier til null ved påtrykk av start ? *)
Referanseglatter_1(r_inn := referanse_til_PID, Ts := samplingstid, referanse_ut => glatt_referanse);
Lead_lag_1(Kf := kfk, Tlead := tau_lead, Tlag := tau_lag, Ts := samplingstid, leadlag := forover_kobling_bit, reset := resettverdier, y_1 := tanknivaa_til_regulator, outflow := utstroom_til_regulator);
Tracking_1(u_t := ut, Ts := samplingstid, T_tracking := tt, last_u := forrige_paadrag_regulator, aw_på := anti_windup_bit, reset := resettverdier, ui := integralledd, u_it => uit);
PID_regulator_1(EN := start OR kritisk_lav_eller_hooy, Ts := samplingstid, ni := d_filter, Kp_reg := Kp, Ti_reg := Ti, Td_reg := Td, r_1 := glatt_referanse, y_1 := tanknivaa_til_regulator, manual_input := manuelt_paadrag_til_regulator, Regulator_type := reg_modus, u_fk := Lead_lag_1.u_fk, u_antiwindup := Tracking_1.u_antiwindup, ratebegrensing := rate_limit, reset := resettverdier, u_it := uit, u_rykkfri := Tracking_1.u_rykkfri, u_nominel := u0_nompaadrag_til_regulator, ui => integralledd, u_ut => paadrag_fra_regulator, last_u => forrige_paadrag_regulator, u_t => ut);
END_PROGRAM

FUNCTION_BLOCK skalering_tanknivaa
VAR_INPUT
  tanknivaa_filtrert_0 : INT;
END_VAR
VAR_OUTPUT
  tanknivaa_til_regulator_1 : REAL;
END_VAR
VAR
  DEROUND_1 : DEROUND;
END_VAR
VAR_OUTPUT
  tanknivaa_skalert_til_scada_0 : INT;
END_VAR
IF (tanknivaa_filtrert_0 < 510) THEN;
	tanknivaa_til_regulator_1 := 0.0;
	tanknivaa_skalert_til_scada_0 := 0;
ELSE
	tanknivaa_til_regulator_1 := INT_TO_REAL(tanknivaa_filtrert_0-510)/9.9;
	DEROUND_1(real_to_round := INT_TO_REAL(tanknivaa_filtrert_0-510)/9.9*100.0, gjelende_siffer_input := 0);
	tanknivaa_skalert_til_scada_0 := REAL_TO_INT(DEROUND_1.real_rounded);
END_IF;
END_FUNCTION_BLOCK

FUNCTION_BLOCK skalering_ventil
VAR_INPUT
  ventil_input : INT;
END_VAR
VAR_OUTPUT
  ventil_regulator : REAL;
  ventil_scada : INT;
END_VAR
VAR
  DEROUND_1 : DEROUND;
END_VAR
DEROUND_1(real_to_round :=  INT_TO_REAL(ventil_input - 500)/0.35, gjelende_siffer_input := 0);
ventil_scada :=  REAL_TO_INT(DEROUND_1.real_rounded);
ventil_regulator := INT_TO_REAL(ventil_input - 500)/35.0;
END_FUNCTION_BLOCK

FUNCTION_BLOCK skalering_paadrag
VAR_INPUT
  paadrag_fra_regulator_0 : REAL;
  paadrag_manuelt_1 : INT;
  u0_nompaadrag_fra_scada_2 : INT;
END_VAR
VAR_OUTPUT
  paadrag_til_scada_0 : INT;
  manuelt_paadrag_til_regulator_3 : REAL;
  u0_nompaadrag_til_regulator_4 : REAL;
END_VAR
VAR
  DEROUND_1 : DEROUND;
  DEROUND_2 : DEROUND;
END_VAR
VAR_OUTPUT
  frekvenspaadrag_til_omformer_1 : INT;
  ventil_paadrag_2 : INT;
END_VAR
VAR
  DEROUND_3 : DEROUND;
END_VAR
IF pumpe_regulering THEN;
	DEROUND_1(real_to_round :=  paadrag_fra_regulator_0*84.85 + 7825.0, gjelende_siffer_input := 0);
	frekvenspaadrag_til_omformer_1 :=  REAL_TO_INT(DEROUND_1.real_rounded);
ELSIF ventil_regulering THEN;
	DEROUND_2(real_to_round :=  paadrag_fra_regulator_0*35.0 + 500.0, gjelende_siffer_input := 0);
	ventil_paadrag_2 := REAL_TO_INT(DEROUND_2.real_rounded);
END_IF;
DEROUND_3(real_to_round :=  paadrag_fra_regulator_0*100.0, gjelende_siffer_input := 0);
paadrag_til_scada_0 :=  REAL_TO_INT(DEROUND_3.real_rounded);
manuelt_paadrag_til_regulator_3 := INT_TO_REAL(paadrag_manuelt_1)/100.0;
u0_nompaadrag_til_regulator_4 := INT_TO_REAL(u0_nompaadrag_fra_scada_2)/100.0;
END_FUNCTION_BLOCK

FUNCTION_BLOCK skalering_referanse
VAR_INPUT
  referanse_0 : INT;
END_VAR
VAR_OUTPUT
  referanse_til_PID_0 : REAL;
  ref_skalert_som_tankmaaling_1 : INT;
END_VAR
VAR
  DEROUND_1 : DEROUND;
END_VAR
VAR_INPUT
  glatt_referanse_1 : REAL;
END_VAR
VAR_OUTPUT
  glatt_referanse_til_scada_2 : INT;
END_VAR
VAR
  DEROUND_2 : DEROUND;
END_VAR
referanse_til_PID_0 :=  INT_TO_REAL(referanse_0)/100.0;
DEROUND_1(real_to_round := referanse_til_PID_0*9.9 + 510.0, gjelende_siffer_input := 0);
ref_skalert_som_tankmaaling_1 :=  REAL_TO_INT(DEROUND_1.real_rounded);
DEROUND_2(real_to_round := glatt_referanse_1*100.0, gjelende_siffer_input := 0);
glatt_referanse_til_scada_2 :=  REAL_TO_INT(DEROUND_2.real_rounded);
END_FUNCTION_BLOCK

FUNCTION_BLOCK utregning_stasjonært_avvik
VAR_INPUT
  ref_skalert_til_tankmaaling_0 : INT;
  tanknivaa_filtrert_1 : INT;
  start_2 : BOOL;
  ack_3 : BOOL;
END_VAR
VAR
  myTimer : TON;
END_VAR
VAR_OUTPUT
  stasjonært_avvik_verdi_0 : INT;
  stasjonært_avvik_1 : BOOL;
END_VAR
stasjonært_avvik_verdi_0 := ABS(ref_skalert_til_tankmaaling_0 - tanknivaa_filtrert_1);

IF ((stasjonært_avvik_verdi_0 >= 99 ) AND (start_2) AND (NOT ack_3))THEN;
	myTimer(IN := TRUE, PT := T#60s);
ELSE
	myTimer(IN := FALSE);
END_IF;

IF myTimer.Q THEN
	stasjonært_avvik_1 := TRUE;
ELSE
	stasjonært_avvik_1 := FALSE;
END_IF;
END_FUNCTION_BLOCK

FUNCTION_BLOCK skalering_til_bruker_ven_og_omf
VAR_INPUT
  frekvenspaadrag_til_omformer_0 : INT;
  aapning_reg_ventil_1 : INT;
END_VAR
VAR_OUTPUT
  frekvens_skalert_0 : INT;
  ventil_skalert_1 : INT;
END_VAR
VAR
  DEROUND_1 : DEROUND;
  DEROUND_2 : DEROUND;
END_VAR
IF frekvenspaadrag_til_omformer_0 < 7825 THEN;
	frekvens_skalert_0 :=  0;
ELSE
	DEROUND_1(real_to_round := (INT_TO_REAL(frekvenspaadrag_til_omformer_0) - 7825.0)/0.8485, gjelende_siffer_input := 0);
	frekvens_skalert_0 :=  REAL_TO_INT(DEROUND_1.real_rounded);
END_IF;
DEROUND_2(real_to_round := (INT_TO_REAL(aapning_reg_ventil_1) - 500.0)/0.35, gjelende_siffer_input := 0);
ventil_skalert_1 := REAL_TO_INT(DEROUND_2.real_rounded);
END_FUNCTION_BLOCK

FUNCTION_BLOCK skalering_utstroom
VAR_INPUT
  utstroom_filtrert_0 : INT;
END_VAR
VAR_OUTPUT
  utstroom_til_regulator_0 : REAL;
END_VAR
VAR
  DEROUND_1 : DEROUND;
END_VAR
VAR_OUTPUT
  utstroom_til_scada_1 : INT;
END_VAR
VAR
  DEROUND_2 : DEROUND;
END_VAR
IF utstroom_filtrert_0 < 400 THEN;
	utstroom_til_regulator_0 := 0.0;
	utstroom_til_scada_1 := 0;
ELSE
	utstroom_til_regulator_0 := INT_TO_REAL(utstroom_filtrert_0-400)/12.35;
	DEROUND_2(real_to_round := INT_TO_REAL(utstroom_filtrert_0 - 400)/200.00, gjelende_siffer_input := 2);
	utstroom_til_scada_1 := REAL_TO_INT(DEROUND_2.real_rounded*100.00);
END_IF;
END_FUNCTION_BLOCK

FUNCTION_BLOCK mottak_av_data_fra_master
VAR_INPUT
  profibusadresse_0 : INT;
  profibusadresse_1 : INT;
  profibusadresse_2 : INT;
  profibusadresse_3 : INT;
  profibusadresse_4 : INT;
  profibusadresse_5 : INT;
  profibusadresse_6 : INT;
  profibusadresse_7 : INT;
  profibusadresse_8 : INT;
  profibusadresse_9 : INT;
  profibusadresse_10 : INT;
  profibusadresse_11 : INT;
  profibusadresse_12 : INT;
  profibusadresse_13 : INT;
  profibusadresse_14 : INT;
  profibusadresse_15 : INT;
END_VAR
VAR_OUTPUT
  mottak_fra_kanal_0 : INT;
  mottak_fra_kanal_1 : INT;
  mottak_fra_kanal_2 : INT;
  mottak_fra_kanal_3 : INT;
  mottak_fra_kanal_4 : INT;
  mottak_fra_kanal_5 : INT;
  mottak_fra_kanal_6 : INT;
  mottak_fra_kanal_7 : INT;
  mottak_fra_kanal_8 : INT;
  mottak_fra_kanal_9 : INT;
  mottak_fra_kanal_10 : INT;
  mottak_fra_kanal_11 : INT;
  mottak_fra_kanal_12 : INT;
  mottak_fra_kanal_13 : INT;
  mottak_fra_kanal_14 : INT;
  mottak_fra_kanal_15 : INT;
END_VAR
(* structured ladder/FBD written out as ST: instructions are called as NAME(EN, inputs, outputs); _pN, _eN, _tN stand for wires *)
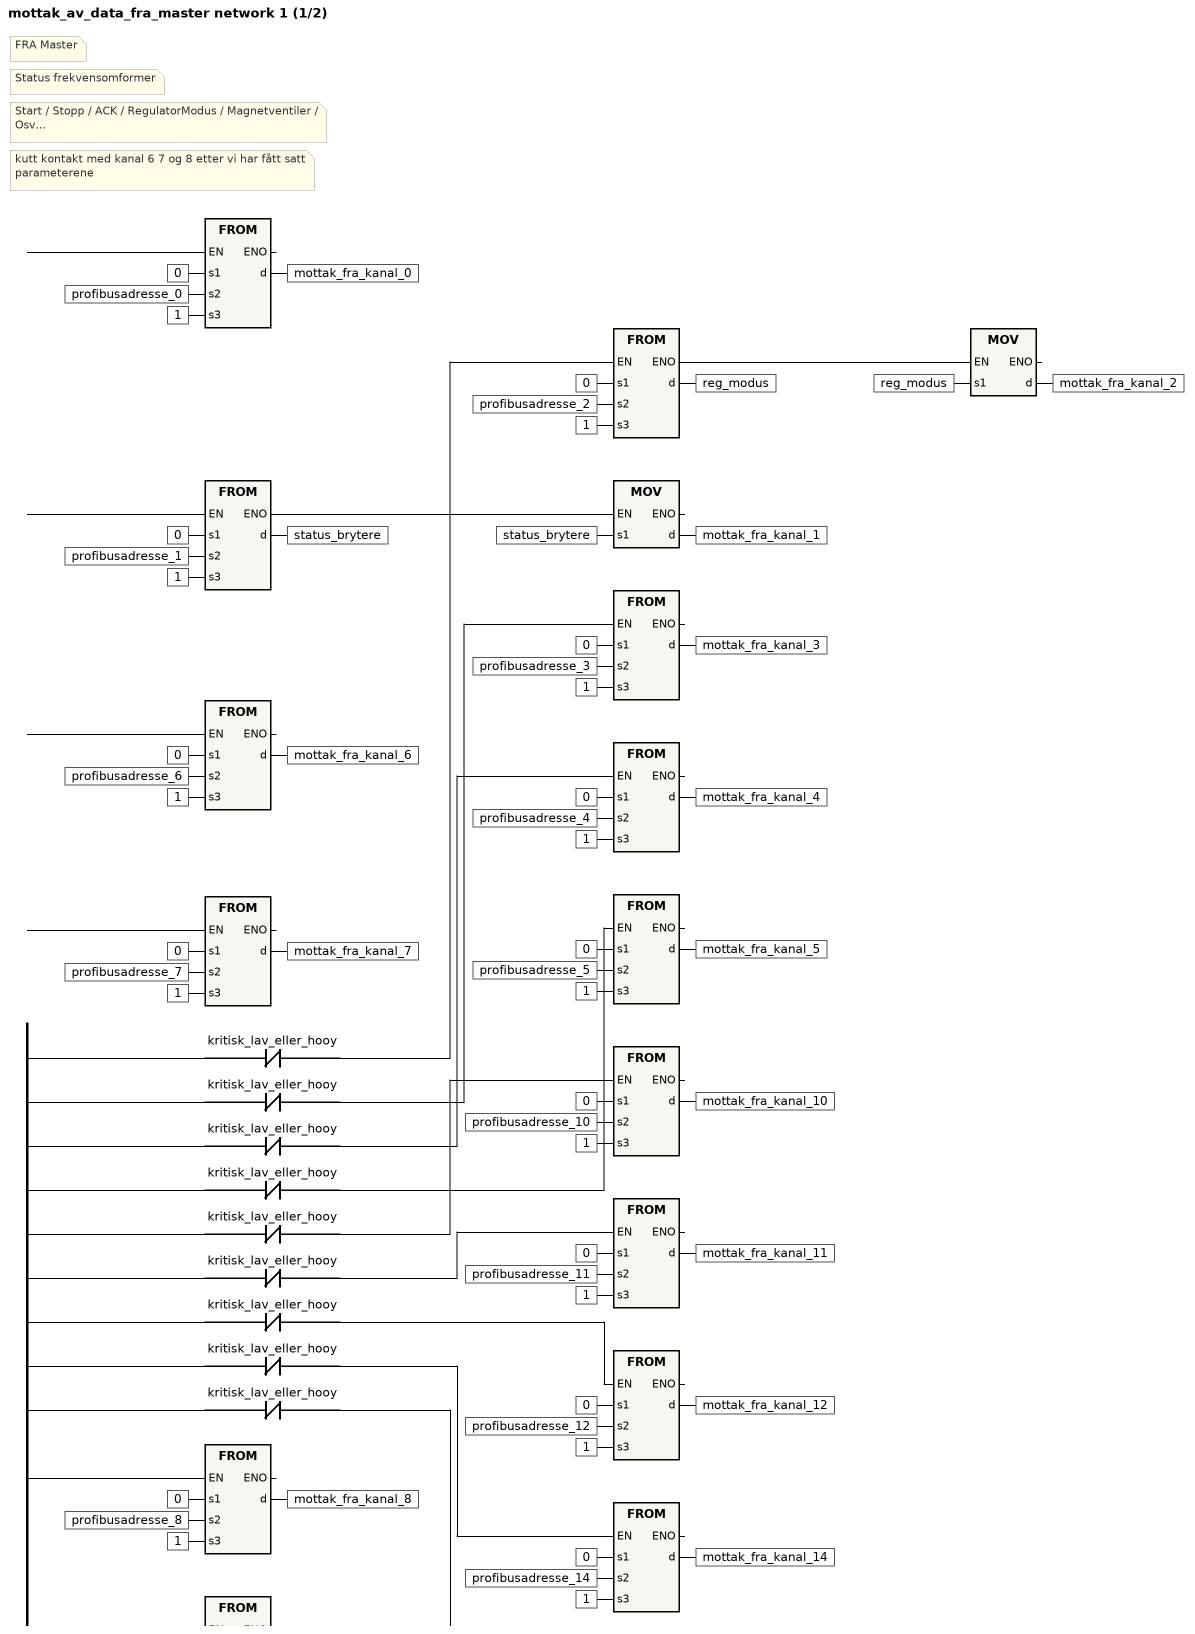
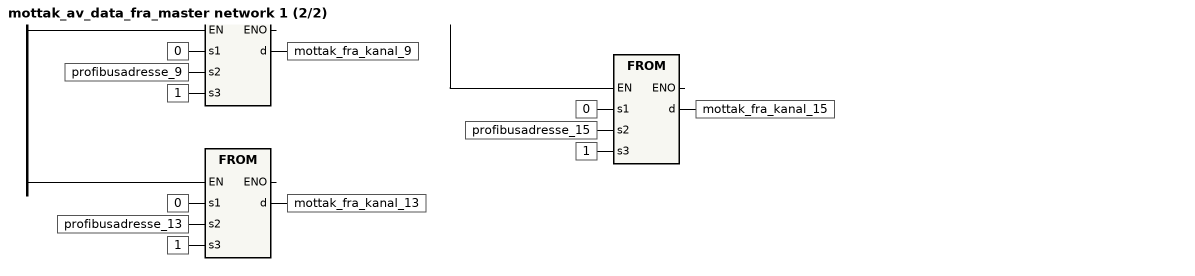
(* network 1 *)
(* FRA Master *)
(* Status frekvensomformer *)
(* Start / Stopp / ACK / RegulatorModus / Magnetventiler / Osv... *)
(* kutt kontakt med kanal 6 7 og 8 etter vi har fått satt parameterene *)
FROM(TRUE, 0, profibusadresse_0, 1, mottak_fra_kanal_0);
_e1 := FROM(TRUE, 0, profibusadresse_1, 1, status_brytere);
MOV(_e1, status_brytere, mottak_fra_kanal_1);
_e2 := FROM(NOT kritisk_lav_eller_hooy, 0, profibusadresse_2, 1, reg_modus);
MOV(_e2, reg_modus, mottak_fra_kanal_2);
FROM(NOT kritisk_lav_eller_hooy, 0, profibusadresse_3, 1, mottak_fra_kanal_3);
FROM(NOT kritisk_lav_eller_hooy, 0, profibusadresse_4, 1, mottak_fra_kanal_4);
FROM(NOT kritisk_lav_eller_hooy, 0, profibusadresse_5, 1, mottak_fra_kanal_5);
FROM(TRUE, 0, profibusadresse_6, 1, mottak_fra_kanal_6);
FROM(TRUE, 0, profibusadresse_7, 1, mottak_fra_kanal_7);
FROM(TRUE, 0, profibusadresse_8, 1, mottak_fra_kanal_8);
FROM(TRUE, 0, profibusadresse_9, 1, mottak_fra_kanal_9);
FROM(NOT kritisk_lav_eller_hooy, 0, profibusadresse_10, 1, mottak_fra_kanal_10);
FROM(NOT kritisk_lav_eller_hooy, 0, profibusadresse_11, 1, mottak_fra_kanal_11);
FROM(NOT kritisk_lav_eller_hooy, 0, profibusadresse_12, 1, mottak_fra_kanal_12);
FROM(TRUE, 0, profibusadresse_13, 1, mottak_fra_kanal_13);
FROM(NOT kritisk_lav_eller_hooy, 0, profibusadresse_14, 1, mottak_fra_kanal_14);
FROM(NOT kritisk_lav_eller_hooy, 0, profibusadresse_15, 1, mottak_fra_kanal_15);
END_FUNCTION_BLOCK

FUNCTION_BLOCK sending_av_data_til_master
VAR_INPUT
  sende_til_kanal_0 : INT;
  sende_til_kanal_1 : INT;
  sende_til_kanal_2 : INT;
  sende_til_kanal_3 : INT;
  sende_til_kanal_4 : INT;
  sende_til_kanal_5 : INT;
  sende_til_kanal_6 : INT;
  sende_til_kanal_7 : INT;
  sende_til_kanal_8 : INT;
  sende_til_kanal_9 : INT;
  sende_til_kanal_10 : INT;
  sende_til_kanal_11 : INT;
  sende_til_kanal_12 : INT;
  sende_til_kanal_13 : INT;
  sende_til_kanal_14 : INT;
  sende_til_kanal_15 : INT;
END_VAR
(* structured ladder/FBD written out as ST: instructions are called as NAME(EN, inputs, outputs); _pN, _eN, _tN stand for wires *)
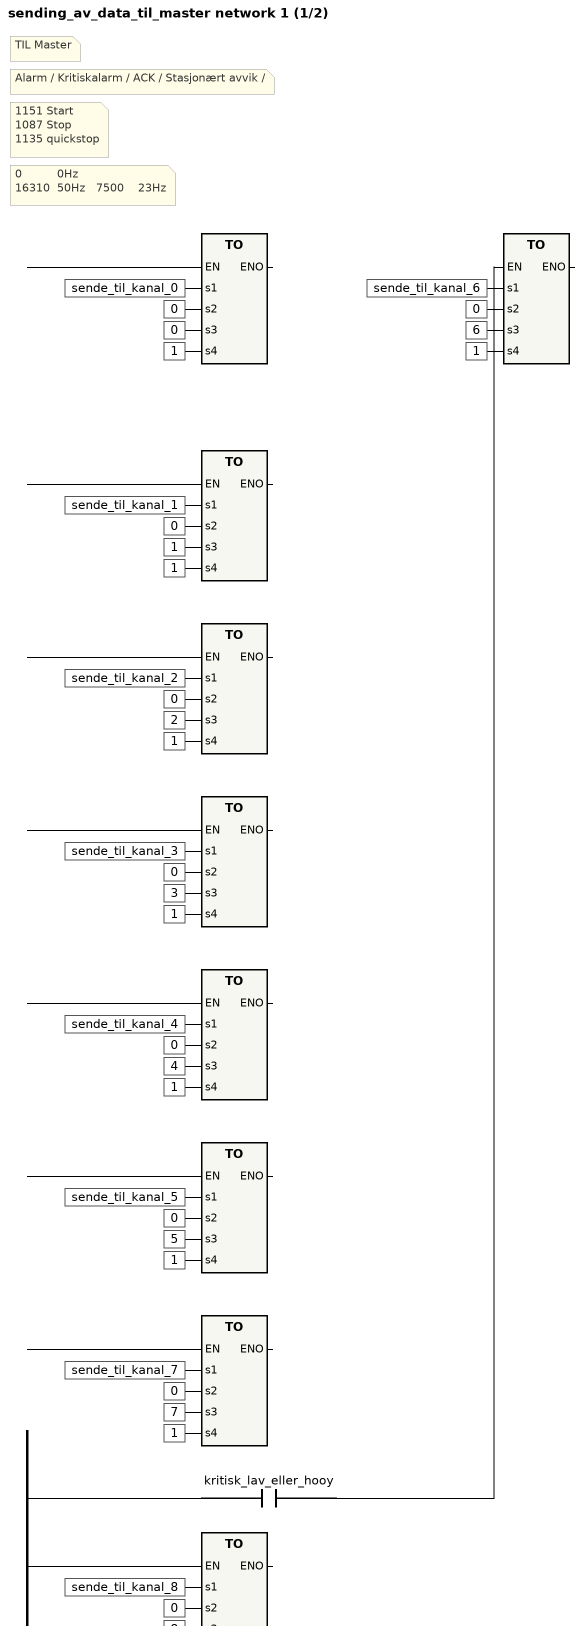
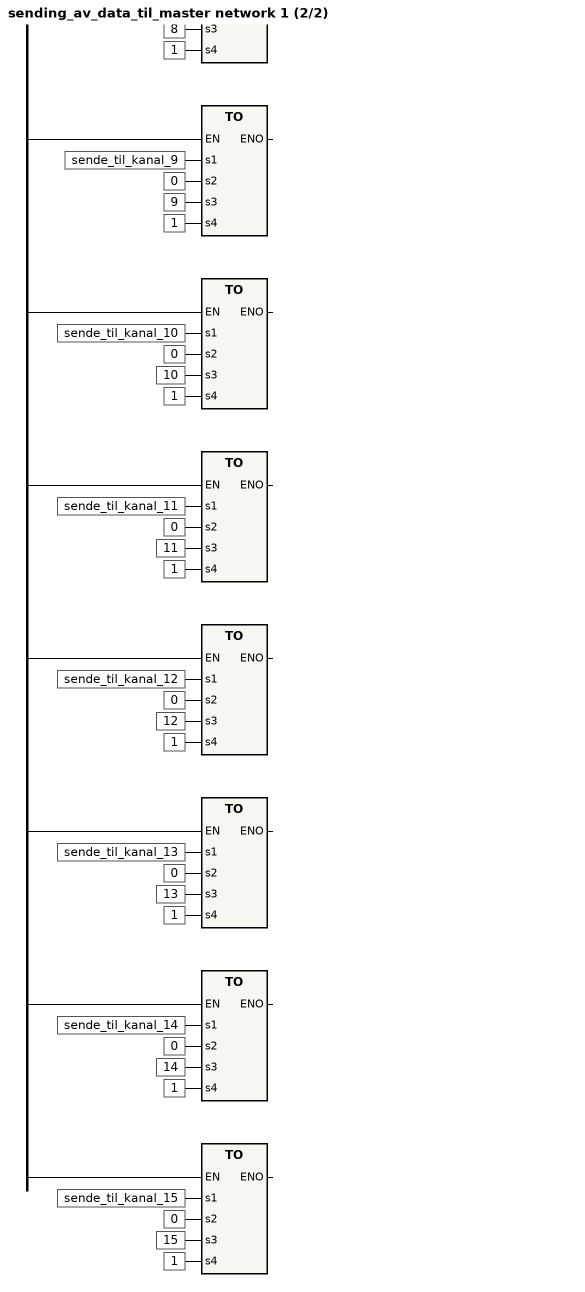
(* network 1 *)
(* TIL Master *)
(* Alarm / Kritiskalarm / ACK / Stasjonært avvik / *)
(* 1151 Start / 1087 Stop / 1135 quickstop *)
(* 0          0Hz / 16310  50Hz   7500    23Hz *)
TO(TRUE, sende_til_kanal_0, 0, 0, 1);
TO(TRUE, sende_til_kanal_1, 0, 1, 1);
TO(TRUE, sende_til_kanal_2, 0, 2, 1);
TO(TRUE, sende_til_kanal_3, 0, 3, 1);
TO(TRUE, sende_til_kanal_4, 0, 4, 1);
TO(TRUE, sende_til_kanal_5, 0, 5, 1);
TO(kritisk_lav_eller_hooy, sende_til_kanal_6, 0, 6, 1);
TO(TRUE, sende_til_kanal_7, 0, 7, 1);
TO(TRUE, sende_til_kanal_8, 0, 8, 1);
TO(TRUE, sende_til_kanal_9, 0, 9, 1);
TO(TRUE, sende_til_kanal_10, 0, 10, 1);
TO(TRUE, sende_til_kanal_11, 0, 11, 1);
TO(TRUE, sende_til_kanal_12, 0, 12, 1);
TO(TRUE, sende_til_kanal_13, 0, 13, 1);
TO(TRUE, sende_til_kanal_14, 0, 14, 1);
TO(TRUE, sende_til_kanal_15, 0, 15, 1);
END_FUNCTION_BLOCK

FUNCTION_BLOCK kvittering_av_alarmer
VAR_INPUT
  ACK_bit_0 : BOOL;
END_VAR
VAR_OUTPUT
  alarm_nedre_1 : BOOL;
  kritiskalarm_oovre_2 : BOOL;
  kritiskalarm_nedre_3 : BOOL;
  alarm_oovre_0 : BOOL;
  strømbrudd_4 : BOOL;
  stasjonært_avvik_5 : BOOL;
  kritiskalarm_refnivaa_oppnaad_6 : BOOL;
  auto_ACK_7 : BOOL;
  auto_ACK_lav_hooy_8 : BOOL;
  ACK_slave_9 : BOOL;
  fortsatt_alarm_10 : BOOL;
  kritisk_refnivaa_opnaad_slave_11 : BOOL;
END_VAR
VAR_INPUT
  kritisk_lav_eller_hooy_1 : BOOL;
END_VAR
(* structured ladder/FBD written out as ST: instructions are called as NAME(EN, inputs, outputs); _pN, _eN, _tN stand for wires *)
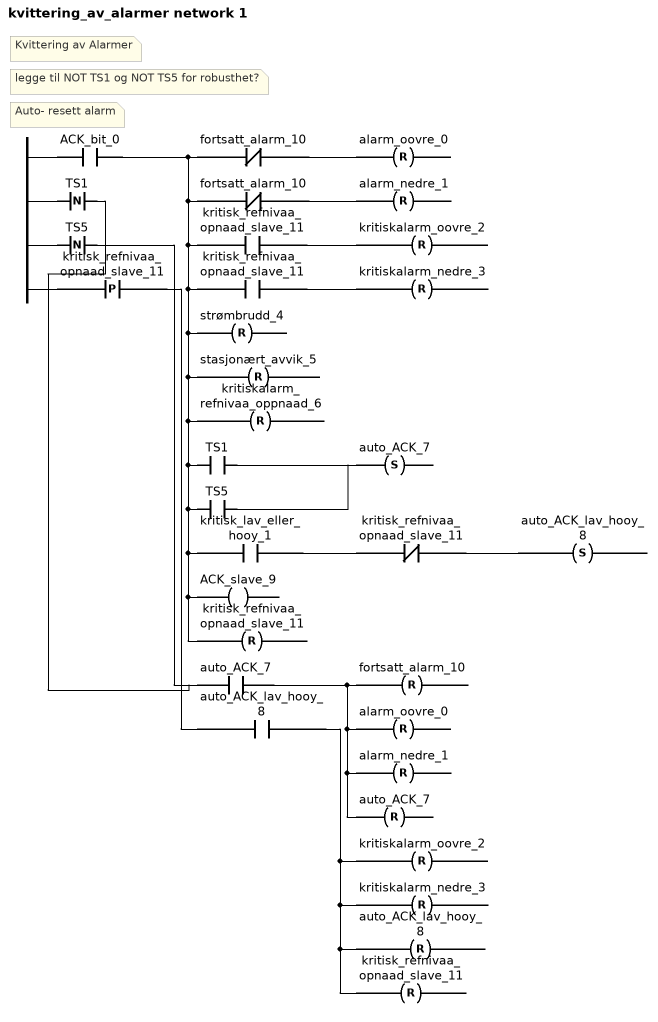
(* network 1 *)
(* Kvittering av Alarmer *)
(* legge til NOT TS1 og NOT TS5 for robusthet? *)
(* Auto- resett alarm *)
RST(ACK_bit_0 AND NOT fortsatt_alarm_10, alarm_oovre_0);
RST(ACK_bit_0 AND NOT fortsatt_alarm_10, alarm_nedre_1);
RST(ACK_bit_0 AND kritisk_refnivaa_opnaad_slave_11, kritiskalarm_oovre_2);
RST(ACK_bit_0 AND kritisk_refnivaa_opnaad_slave_11, kritiskalarm_nedre_3);
RST(ACK_bit_0, strømbrudd_4);
RST(ACK_bit_0, stasjonært_avvik_5);
RST(ACK_bit_0, kritiskalarm_refnivaa_oppnaad_6);
SET((ACK_bit_0 AND TS1) OR (ACK_bit_0 AND TS5), auto_ACK_7);
SET(ACK_bit_0 AND kritisk_lav_eller_hooy_1 AND NOT kritisk_refnivaa_opnaad_slave_11, auto_ACK_lav_hooy_8);
ACK_slave_9 := ACK_bit_0;
RST(ACK_bit_0, kritisk_refnivaa_opnaad_slave_11);
_p1 := (LDF(TRUE, TS1) OR LDF(TRUE, TS5)) AND auto_ACK_7;
RST(_p1, fortsatt_alarm_10);
RST(_p1, alarm_oovre_0);
RST(_p1, alarm_nedre_1);
RST(_p1, auto_ACK_7);
_p2 := LDP(TRUE, kritisk_refnivaa_opnaad_slave_11) AND auto_ACK_lav_hooy_8;
RST(_p2, kritiskalarm_oovre_2);
RST(_p2, kritiskalarm_nedre_3);
RST(_p2, auto_ACK_lav_hooy_8);
RST(_p2, kritisk_refnivaa_opnaad_slave_11);
END_FUNCTION_BLOCK

FUNCTION_BLOCK utganger
VAR_INPUT
  tvangstyr_startsignal_frekv_0 : BOOL;
END_VAR
VAR_OUTPUT
  fysisk_start_frekomformer_0 : BOOL;
  magnetventil_1_1 : BOOL;
  magnetventil_2_2 : BOOL;
  magnetventil_3_3 : BOOL;
  magnetventil_1_ACK_4 : BOOL;
  magnetventil_2_ACK_5 : BOOL;
  magnetventil_3_ACK_6 : BOOL;
END_VAR
VAR_INPUT
  aktiver_magv_1_bit_1 : BOOL;
  aktiver_magv_2_bit_2 : BOOL;
  aktiver_magv_3_bit_3 : BOOL;
  kritiaskalarm_aapne_ventiler_4 : BOOL;
  kritisk_refnivaa_opnaad_slave_5 : BOOL;
  kritiskalarm_nedre_stengventil_6 : BOOL;
  under_60_nivaa_7 : BOOL;
END_VAR
(* structured ladder/FBD written out as ST: instructions are called as NAME(EN, inputs, outputs); _pN, _eN, _tN stand for wires *)
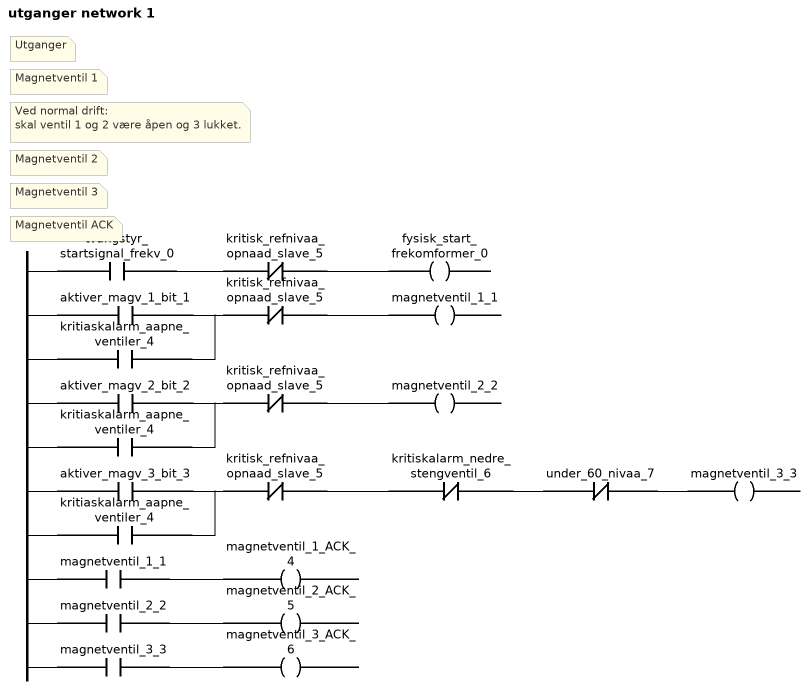
(* network 1 *)
(* Utganger *)
(* Magnetventil 1 *)
(* Ved normal drift: / skal ventil 1 og 2 være åpen og 3 lukket. *)
(* Magnetventil 2 *)
(* Magnetventil 3 *)
(* Magnetventil ACK *)
fysisk_start_frekomformer_0 := tvangstyr_startsignal_frekv_0 AND NOT kritisk_refnivaa_opnaad_slave_5;
magnetventil_1_1 := (aktiver_magv_1_bit_1 OR kritiaskalarm_aapne_ventiler_4) AND NOT kritisk_refnivaa_opnaad_slave_5;
magnetventil_2_2 := (aktiver_magv_2_bit_2 OR kritiaskalarm_aapne_ventiler_4) AND NOT kritisk_refnivaa_opnaad_slave_5;
magnetventil_3_3 := (((aktiver_magv_3_bit_3 OR kritiaskalarm_aapne_ventiler_4) AND NOT kritisk_refnivaa_opnaad_slave_5) AND NOT kritiskalarm_nedre_stengventil_6) AND NOT under_60_nivaa_7;
magnetventil_1_ACK_4 := magnetventil_1_1;
magnetventil_2_ACK_5 := magnetventil_2_2;
magnetventil_3_ACK_6 := magnetventil_3_3;
END_FUNCTION_BLOCK

FUNCTION_BLOCK reguleringsmodus
VAR_INPUT
  pumpe_regulering_bit_0 : BOOL;
END_VAR
VAR_OUTPUT
  pumpe_regulering_0 : BOOL;
  ventil_regulering_1 : BOOL;
END_VAR
VAR_INPUT
  ventil_regulering_bit_1 : BOOL;
  ventil_paadrag_2 : INT;
END_VAR
VAR_OUTPUT
  aapning_reg_ventil_2 : INT;
  frekvenspaadrag_til_omformer_3 : INT;
END_VAR
VAR_INPUT
  start_3 : BOOL;
END_VAR
(* structured ladder/FBD written out as ST: instructions are called as NAME(EN, inputs, outputs); _pN, _eN, _tN stand for wires *)
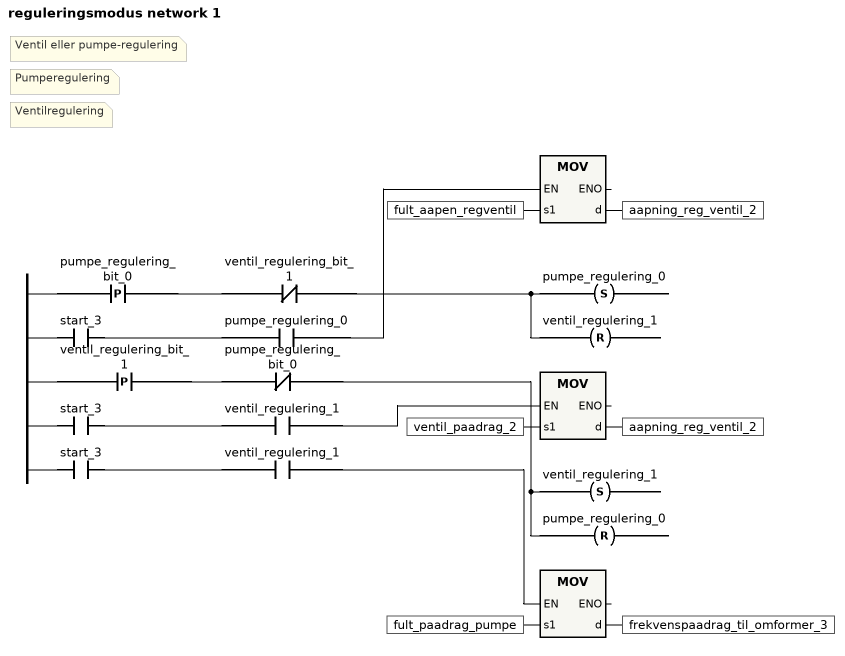
(* network 1 *)
(* Ventil eller pumpe-regulering *)
(* Pumperegulering *)
(* Ventilregulering *)
_p1 := LDP(TRUE, pumpe_regulering_bit_0) AND NOT ventil_regulering_bit_1;
SET(_p1, pumpe_regulering_0);
RST(_p1, ventil_regulering_1);
MOV(start_3 AND pumpe_regulering_0, fult_aapen_regventil, aapning_reg_ventil_2);
_p2 := LDP(TRUE, ventil_regulering_bit_1) AND NOT pumpe_regulering_bit_0;
SET(_p2, ventil_regulering_1);
RST(_p2, pumpe_regulering_0);
MOV(start_3 AND ventil_regulering_1, ventil_paadrag_2, aapning_reg_ventil_2);
MOV(start_3 AND ventil_regulering_1, fult_paadrag_pumpe, frekvenspaadrag_til_omformer_3);
END_FUNCTION_BLOCK

FUNCTION_BLOCK kritisk_refnivaa_oppnaad
VAR_INPUT
  innenfor_refomraade_0 : BOOL;
  kritisk_lav_eller_hooy_1 : BOOL;
END_VAR
VAR_OUTPUT
  kritisk_refnivaa_opnaad_slave_0 : BOOL;
  kritiskalarm_refnivaa_oppnaad_1 : BOOL;
  frekvenspaadrag_til_omformer_2 : INT;
  control_word_3 : INT;
  aapning_reg_ventil_4 : INT;
END_VAR
(* structured ladder/FBD written out as ST: instructions are called as NAME(EN, inputs, outputs); _pN, _eN, _tN stand for wires *)
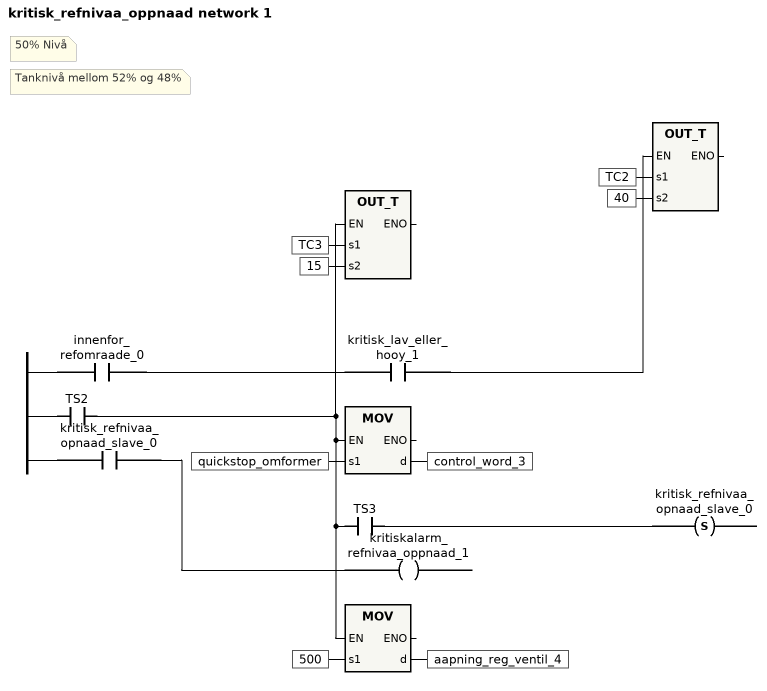
(* network 1 *)
(* 50% Nivå *)
(* Tanknivå mellom 52% og 48% *)
OUT_T(innenfor_refomraade_0 AND kritisk_lav_eller_hooy_1, TC2, 40);
OUT_T(TS2, TC3, 15);
SET(TS2 AND TS3, kritisk_refnivaa_opnaad_slave_0);
MOV(TS2, quickstop_omformer, control_word_3);
MOV(TS2, 500, aapning_reg_ventil_4);
kritiskalarm_refnivaa_oppnaad_1 := kritisk_refnivaa_opnaad_slave_0;
END_FUNCTION_BLOCK

FUNCTION_BLOCK handling_ved_kritisk_alarm
VAR_INPUT
  kritiskalarm_oovre_0 : BOOL;
  kritiskalarm_nedre_1 : BOOL;
END_VAR
VAR_OUTPUT
  referanse_0 : INT;
  reg_modus_1 : INT;
  u0_nompaadrag_fra_scada_2 : INT;
END_VAR
VAR_INPUT
  tanknivaa_filtrert_2 : INT;
END_VAR
VAR_OUTPUT
  under_60_nivaa_3 : BOOL;
END_VAR
(* structured ladder/FBD written out as ST: instructions are called as NAME(EN, inputs, outputs); _pN, _eN, _tN stand for wires *)
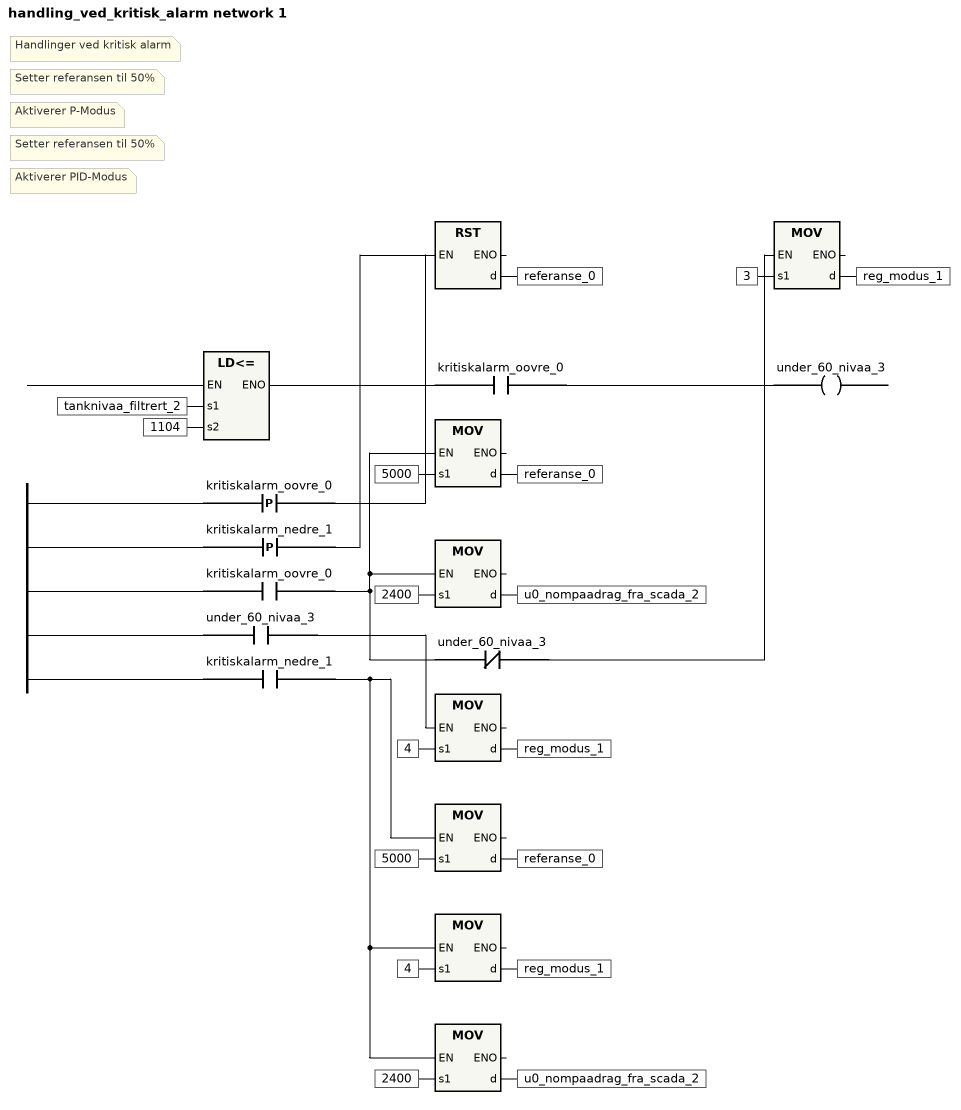
(* network 1 *)
(* Handlinger ved kritisk alarm *)
(* Setter referansen til 50% *)
(* Aktiverer P-Modus *)
(* Setter referansen til 50% *)
(* Aktiverer PID-Modus *)
RST(LDP(TRUE, kritiskalarm_oovre_0) OR LDP(TRUE, kritiskalarm_nedre_1), referanse_0);
MOV(kritiskalarm_oovre_0, 5000, referanse_0);
MOV(kritiskalarm_oovre_0 AND NOT under_60_nivaa_3, 3, reg_modus_1);
MOV(kritiskalarm_oovre_0, 2400, u0_nompaadrag_fra_scada_2);
_e1 := LD<=(TRUE, tanknivaa_filtrert_2, 1104);
under_60_nivaa_3 := _e1 AND kritiskalarm_oovre_0;
MOV(under_60_nivaa_3, 4, reg_modus_1);
MOV(kritiskalarm_nedre_1, 5000, referanse_0);
MOV(kritiskalarm_nedre_1, 4, reg_modus_1);
MOV(kritiskalarm_nedre_1, 2400, u0_nompaadrag_fra_scada_2);
END_FUNCTION_BLOCK

FUNCTION_BLOCK alarmgrenser
VAR_OUTPUT
  kritiskalarm_oovre_0 : BOOL;
  kritiskalarm_nedre_1 : BOOL;
  kritisk_lav_eller_hooy_2 : BOOL;
  alarm_oovre_3 : BOOL;
  alarm_nedre_4 : BOOL;
END_VAR
VAR_INPUT
  start_0 : BOOL;
  ACK_bit_1 : BOOL;
  tanknivaa_filtrert_2 : INT;
END_VAR
VAR_OUTPUT
  fortsatt_alarm_5 : BOOL;
END_VAR
(* structured ladder/FBD written out as ST: instructions are called as NAME(EN, inputs, outputs); _pN, _eN, _tN stand for wires *)
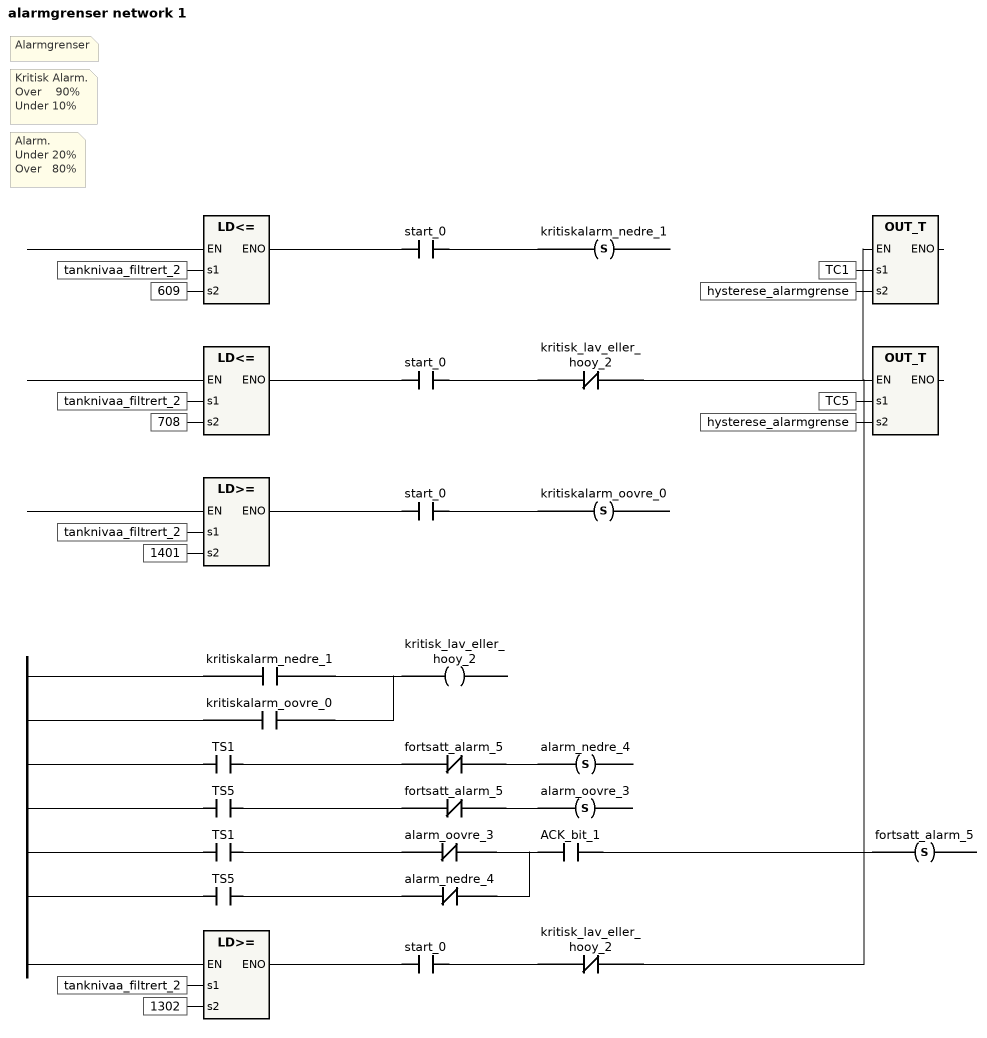
(* network 1 *)
(* Alarmgrenser *)
(* Kritisk Alarm. /  / Over    90% / Under 10% *)
(* Alarm. /  / Under 20% / Over   80% *)
_e1 := LD<=(TRUE, tanknivaa_filtrert_2, 609);
SET(_e1 AND start_0, kritiskalarm_nedre_1);
_e2 := LD>=(TRUE, tanknivaa_filtrert_2, 1401);
SET(_e2 AND start_0, kritiskalarm_oovre_0);
kritisk_lav_eller_hooy_2 := kritiskalarm_nedre_1 OR kritiskalarm_oovre_0;
_e3 := LD<=(TRUE, tanknivaa_filtrert_2, 708);
OUT_T(_e3 AND start_0 AND NOT kritisk_lav_eller_hooy_2, TC1, hysterese_alarmgrense);
_e4 := LD>=(TRUE, tanknivaa_filtrert_2, 1302);
OUT_T(_e4 AND start_0 AND NOT kritisk_lav_eller_hooy_2, TC5, hysterese_alarmgrense);
SET(TS1 AND NOT fortsatt_alarm_5, alarm_nedre_4);
SET(TS5 AND NOT fortsatt_alarm_5, alarm_oovre_3);
SET(((TS1 AND NOT alarm_oovre_3) OR (TS5 AND NOT alarm_nedre_4)) AND ACK_bit_1, fortsatt_alarm_5);
END_FUNCTION_BLOCK

FUNCTION_BLOCK lavpass_filter_utstrøm
VAR CONSTANT
  omega_0 : REAL := 0.2;  (* cutoff frekvens. 16.4: 0.25 mye støy?? gamle:0.0384 *)
  two_pi : REAL := 6.28;  (* 2*pi *)
END_VAR
VAR_INPUT
  samplingstid_0 : INT;
END_VAR
VAR_OUTPUT
  utstroom_filtrert_0 : INT;
END_VAR
VAR
  DEROUND_1 : DEROUND;
END_VAR
VAR_INPUT
  utstroom_analogt_1 : INT;
END_VAR
VAR
  input_float : REAL;
  avg_maaling : REAL;
  avg_maaling_k_minus_1 : REAL;
  filter_faktor : REAL;
  eksponent : REAL;
  tastetid_float : REAL;
END_VAR
tastetid_float :=  INT_TO_REAL (samplingstid_0)/100.0;
eksponent := -tastetid_float*omega_0*two_pi;
filter_faktor := EXP(eksponent);
input_float := INT_TO_REAL (utstroom_analogt_1);
avg_maaling := filter_faktor * avg_maaling_k_minus_1 + (1.0 - filter_faktor) * input_float;
avg_maaling_k_minus_1 := avg_maaling;
DEROUND_1(real_to_round := avg_maaling, gjelende_siffer_input := 0);
utstroom_filtrert_0 := REAL_TO_INT(DEROUND_1.real_rounded);
END_FUNCTION_BLOCK

PROGRAM stroombrudd
(* structured ladder/FBD written out as ST: instructions are called as NAME(EN, inputs, outputs); _pN, _eN, _tN stand for wires *)
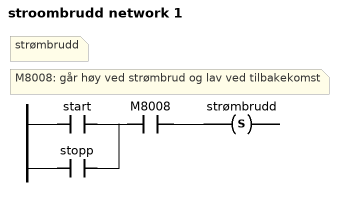
(* network 1 *)
(* strømbrudd *)
(* M8008: går høy ved strømbrud og lav ved tilbakekomst *)
SET((start OR stopp) AND M8008, strømbrudd);
END_PROGRAM
